KUKA KRL program: rebar_install.src

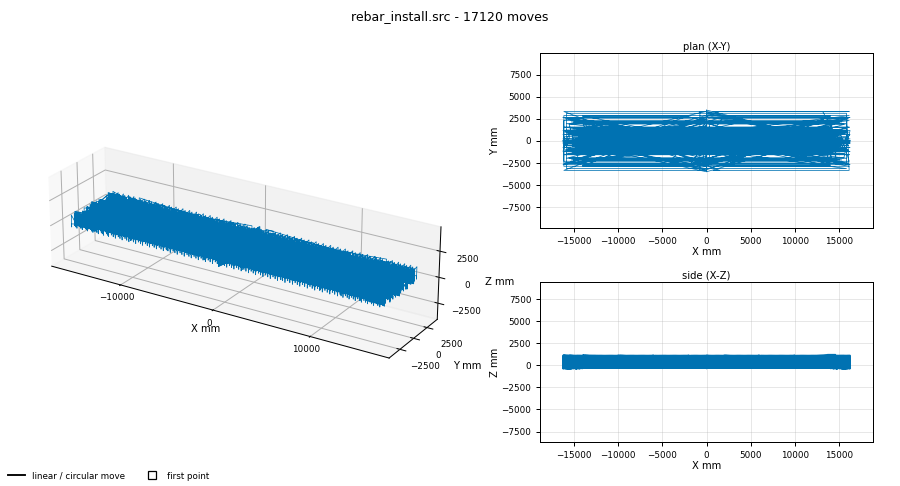
[picture p0: tool path of rebar_install.src, 17120 of 17120 moves have a stored position in this frame; points joined in program order, loops and branches not executed]
&ACCESS RVP
&REL 1
DEF REBAR_INSTALL()
  BAS(#INITMOV,0)
  ; Step 1, bar 1959
  LIN {X 14090.487,Y -1470.303,Z 792.693,A -175.02391,B 0.00000,C -180.00000} ; outside
  LIN {X 14090.487,Y -1470.303,Z -163.061,A -175.02391,B 0.00000,C -180.00000} ; preinsert
  LIN {X 14090.487,Y -1470.303,Z -413.061,A -175.02391,B 0.00000,C -180.00000} ; insert
  LIN {X 14090.487,Y -1470.303,Z -413.061,A -175.02391,B 0.00000,C -180.00000} ; release
  LIN {X 14090.487,Y -1470.303,Z -113.061,A -175.02391,B 0.00000,C -180.00000} ; retreat
  ; Step 2, bar 1960
  LIN {X 14090.487,Y 1470.303,Z 792.693,A 175.02391,B 0.00000,C 180.00000} ; outside
  LIN {X 14090.487,Y 1470.303,Z -163.061,A 175.02391,B 0.00000,C 180.00000} ; preinsert
  LIN {X 14090.487,Y 1470.303,Z -413.061,A 175.02391,B 0.00000,C 180.00000} ; insert
  LIN {X 14090.487,Y 1470.303,Z -413.061,A 175.02391,B 0.00000,C 180.00000} ; release
  LIN {X 14090.487,Y 1470.303,Z -113.061,A 175.02391,B 0.00000,C 180.00000} ; retreat
  ; Step 3, bar 1961
  LIN {X -14090.487,Y -1470.303,Z 792.693,A -4.97609,B 0.00000,C 180.00000} ; outside
  LIN {X -14090.487,Y -1470.303,Z -163.061,A -4.97609,B 0.00000,C 180.00000} ; preinsert
  LIN {X -14090.487,Y -1470.303,Z -413.061,A -4.97609,B 0.00000,C 180.00000} ; insert
  LIN {X -14090.487,Y -1470.303,Z -413.061,A -4.97609,B 0.00000,C 180.00000} ; release
  LIN {X -14090.487,Y -1470.303,Z -113.061,A -4.97609,B 0.00000,C 180.00000} ; retreat
  ; Step 4, bar 1962
  LIN {X -14090.487,Y 1470.303,Z 792.693,A 4.97609,B 0.00000,C 180.00000} ; outside
  LIN {X -14090.487,Y 1470.303,Z -163.061,A 4.97609,B 0.00000,C 180.00000} ; preinsert
  LIN {X -14090.487,Y 1470.303,Z -413.061,A 4.97609,B 0.00000,C 180.00000} ; insert
  LIN {X -14090.487,Y 1470.303,Z -413.061,A 4.97609,B 0.00000,C 180.00000} ; release
  LIN {X -14090.487,Y 1470.303,Z -113.061,A 4.97609,B 0.00000,C 180.00000} ; retreat
  ; Step 5, bar 1954
  LIN {X 0.000,Y -1540.000,Z 792.630,A 0.00000,B 0.00000,C 180.00000} ; outside
  LIN {X 0.000,Y -1540.000,Z -156.000,A 0.00000,B 0.00000,C 180.00000} ; preinsert
  LIN {X 0.000,Y -1540.000,Z -406.000,A 0.00000,B 0.00000,C 180.00000} ; insert
  LIN {X 0.000,Y -1540.000,Z -406.000,A 0.00000,B 0.00000,C 180.00000} ; release
  LIN {X 0.000,Y -1540.000,Z -106.000,A 0.00000,B 0.00000,C 180.00000} ; retreat
  ; Step 6, bar 1949
  LIN {X 0.000,Y 1540.000,Z 792.630,A 0.00000,B 0.00000,C 180.00000} ; outside
  LIN {X 0.000,Y 1540.000,Z -156.000,A 0.00000,B 0.00000,C 180.00000} ; preinsert
  LIN {X 0.000,Y 1540.000,Z -406.000,A 0.00000,B 0.00000,C 180.00000} ; insert
  LIN {X 0.000,Y 1540.000,Z -406.000,A 0.00000,B 0.00000,C 180.00000} ; release
  LIN {X 0.000,Y 1540.000,Z -106.000,A 0.00000,B 0.00000,C 180.00000} ; retreat
  ; Step 7, bar 1859
  LIN {X 0.000,Y -1752.282,Z 792.630,A 0.00000,B 0.00000,C 180.00000} ; outside
  LIN {X 0.000,Y -1752.282,Z -151.145,A 0.00000,B 0.00000,C 180.00000} ; preinsert
  LIN {X 0.000,Y -1752.282,Z -401.145,A 0.00000,B 0.00000,C 180.00000} ; insert
  LIN {X 0.000,Y -1752.282,Z -401.145,A 0.00000,B 0.00000,C 180.00000} ; release
  LIN {X 0.000,Y -1752.282,Z -101.145,A 0.00000,B 0.00000,C 180.00000} ; retreat
  ; Step 8, bar 1926
  LIN {X 0.000,Y -1632.282,Z 792.630,A 0.00000,B 0.00000,C 180.00000} ; outside
  LIN {X 0.000,Y -1632.282,Z -151.145,A 0.00000,B 0.00000,C 180.00000} ; preinsert
  LIN {X 0.000,Y -1632.282,Z -401.145,A 0.00000,B 0.00000,C 180.00000} ; insert
  LIN {X 0.000,Y -1632.282,Z -401.145,A 0.00000,B 0.00000,C 180.00000} ; release
  LIN {X 0.000,Y -1632.282,Z -101.145,A 0.00000,B 0.00000,C 180.00000} ; retreat
  ; Step 9, bar 1925
  LIN {X 0.000,Y 1632.282,Z 792.630,A 0.00000,B 0.00000,C 180.00000} ; outside
  LIN {X 0.000,Y 1632.282,Z -151.145,A 0.00000,B 0.00000,C 180.00000} ; preinsert
  LIN {X 0.000,Y 1632.282,Z -401.145,A 0.00000,B 0.00000,C 180.00000} ; insert
  LIN {X 0.000,Y 1632.282,Z -401.145,A 0.00000,B 0.00000,C 180.00000} ; release
  LIN {X 0.000,Y 1632.282,Z -101.145,A 0.00000,B 0.00000,C 180.00000} ; retreat
  ; Step 10, bar 1872
  LIN {X 0.000,Y 1752.282,Z 792.630,A 0.00000,B 0.00000,C 180.00000} ; outside
  LIN {X 0.000,Y 1752.282,Z -151.145,A 0.00000,B 0.00000,C 180.00000} ; preinsert
  LIN {X 0.000,Y 1752.282,Z -401.145,A 0.00000,B 0.00000,C 180.00000} ; insert
  LIN {X 0.000,Y 1752.282,Z -401.145,A 0.00000,B 0.00000,C 180.00000} ; release
  LIN {X 0.000,Y 1752.282,Z -101.145,A 0.00000,B 0.00000,C 180.00000} ; retreat
  ; Step 11, bar 3422
  LIN {X -16169.500,Y -1557.401,Z 792.630,A 90.00000,B 0.00000,C 180.00000} ; outside
  LIN {X -16169.500,Y -1557.401,Z -142.000,A 90.00000,B 0.00000,C 180.00000} ; preinsert
  LIN {X -16169.500,Y -1557.401,Z -392.000,A 90.00000,B 0.00000,C 180.00000} ; insert
  LIN {X -16169.500,Y -1557.401,Z -392.000,A 90.00000,B 0.00000,C 180.00000} ; release
  LIN {X -16169.500,Y -1557.401,Z -92.000,A 90.00000,B 0.00000,C 180.00000} ; retreat
  ; Step 12, bar 3418
  LIN {X 16169.500,Y -1557.401,Z 792.630,A 90.00000,B 0.00000,C 180.00000} ; outside
  LIN {X 16169.500,Y -1557.401,Z -142.000,A 90.00000,B 0.00000,C 180.00000} ; preinsert
  LIN {X 16169.500,Y -1557.401,Z -392.000,A 90.00000,B 0.00000,C 180.00000} ; insert
  LIN {X 16169.500,Y -1557.401,Z -392.000,A 90.00000,B 0.00000,C 180.00000} ; release
  LIN {X 16169.500,Y -1557.401,Z -92.000,A 90.00000,B 0.00000,C 180.00000} ; retreat
  ; Step 13, bar 3420
  LIN {X -16169.500,Y 1557.401,Z 792.630,A -90.00000,B 0.00000,C 180.00000} ; outside
  LIN {X -16169.500,Y 1557.401,Z -142.000,A -90.00000,B 0.00000,C 180.00000} ; preinsert
  LIN {X -16169.500,Y 1557.401,Z -392.000,A -90.00000,B 0.00000,C 180.00000} ; insert
  LIN {X -16169.500,Y 1557.401,Z -392.000,A -90.00000,B 0.00000,C 180.00000} ; release
  LIN {X -16169.500,Y 1557.401,Z -92.000,A -90.00000,B 0.00000,C 180.00000} ; retreat
  ; Step 14, bar 3416
  LIN {X 16169.500,Y 1557.401,Z 792.630,A -90.00000,B 0.00000,C 180.00000} ; outside
  LIN {X 16169.500,Y 1557.401,Z -142.000,A -90.00000,B 0.00000,C 180.00000} ; preinsert
  LIN {X 16169.500,Y 1557.401,Z -392.000,A -90.00000,B 0.00000,C 180.00000} ; insert
  LIN {X 16169.500,Y 1557.401,Z -392.000,A -90.00000,B 0.00000,C 180.00000} ; release
  LIN {X 16169.500,Y 1557.401,Z -92.000,A -90.00000,B 0.00000,C 180.00000} ; retreat
  ; Step 15, bar 1860
  LIN {X 0.000,Y -1977.000,Z 792.630,A 0.00000,B 0.00000,C 180.00000} ; outside
  LIN {X 0.000,Y -1977.000,Z -124.093,A 0.00000,B 0.00000,C 180.00000} ; preinsert
  LIN {X 0.000,Y -1977.000,Z -374.093,A 0.00000,B 0.00000,C 180.00000} ; insert
  LIN {X 0.000,Y -1977.000,Z -374.093,A 0.00000,B 0.00000,C 180.00000} ; release
  LIN {X 0.000,Y -1977.000,Z -74.093,A 0.00000,B 0.00000,C 180.00000} ; retreat
  ; Step 16, bar 1873
  LIN {X 0.000,Y 1977.000,Z 792.630,A 0.00000,B 0.00000,C 180.00000} ; outside
  LIN {X 0.000,Y 1977.000,Z -124.093,A 0.00000,B 0.00000,C 180.00000} ; preinsert
  LIN {X 0.000,Y 1977.000,Z -374.093,A 0.00000,B 0.00000,C 180.00000} ; insert
  LIN {X 0.000,Y 1977.000,Z -374.093,A 0.00000,B 0.00000,C 180.00000} ; release
  LIN {X 0.000,Y 1977.000,Z -74.093,A 0.00000,B 0.00000,C 180.00000} ; retreat
  ; Step 17, bar 1953
  LIN {X 0.000,Y -1420.000,Z 792.630,A 0.00000,B 0.00000,C 180.00000} ; outside
  LIN {X 0.000,Y -1420.000,Z -118.500,A 0.00000,B 0.00000,C 180.00000} ; preinsert
  LIN {X 0.000,Y -1420.000,Z -368.500,A 0.00000,B 0.00000,C 180.00000} ; insert
  LIN {X 0.000,Y -1420.000,Z -368.500,A 0.00000,B 0.00000,C 180.00000} ; release
  LIN {X 0.000,Y -1420.000,Z -68.500,A 0.00000,B 0.00000,C 180.00000} ; retreat
  ; Step 18, bar 1948
  LIN {X 0.000,Y 1420.000,Z 792.630,A 0.00000,B 0.00000,C 180.00000} ; outside
  LIN {X 0.000,Y 1420.000,Z -118.500,A 0.00000,B 0.00000,C 180.00000} ; preinsert
  LIN {X 0.000,Y 1420.000,Z -368.500,A 0.00000,B 0.00000,C 180.00000} ; insert
  LIN {X 0.000,Y 1420.000,Z -368.500,A 0.00000,B 0.00000,C 180.00000} ; release
  LIN {X 0.000,Y 1420.000,Z -68.500,A 0.00000,B 0.00000,C 180.00000} ; retreat
  ; Step 19, bar 3289
  LIN {X -15485.187,Y -1114.878,Z 792.759,A -134.96824,B 0.00000,C -180.00000} ; outside
  LIN {X -15485.187,Y -1114.878,Z -98.768,A -134.96824,B 0.00000,C -180.00000} ; preinsert
  LIN {X -15485.187,Y -1114.878,Z -348.768,A -134.96824,B 0.00000,C -180.00000} ; insert
  LIN {X -15485.187,Y -1114.878,Z -348.768,A -134.96824,B 0.00000,C -180.00000} ; release
  LIN {X -15485.187,Y -1114.878,Z -48.768,A -134.96824,B 0.00000,C -180.00000} ; retreat
  ; Step 20, bar 3291
  LIN {X -15614.813,Y -1114.878,Z 792.759,A -45.03176,B 0.00000,C 180.00000} ; outside
  LIN {X -15614.813,Y -1114.878,Z -98.768,A -45.03176,B 0.00000,C 180.00000} ; preinsert
  LIN {X -15614.813,Y -1114.878,Z -348.768,A -45.03176,B 0.00000,C 180.00000} ; insert
  LIN {X -15614.813,Y -1114.878,Z -348.768,A -45.03176,B 0.00000,C 180.00000} ; release
  LIN {X -15614.813,Y -1114.878,Z -48.768,A -45.03176,B 0.00000,C 180.00000} ; retreat
  ; Step 21, bar 3369
  LIN {X 15485.187,Y -1114.878,Z 792.759,A -45.03176,B 0.00000,C 180.00000} ; outside
  LIN {X 15485.187,Y -1114.878,Z -98.768,A -45.03176,B 0.00000,C 180.00000} ; preinsert
  LIN {X 15485.187,Y -1114.878,Z -348.768,A -45.03176,B 0.00000,C 180.00000} ; insert
  LIN {X 15485.187,Y -1114.878,Z -348.768,A -45.03176,B 0.00000,C 180.00000} ; release
  LIN {X 15485.187,Y -1114.878,Z -48.768,A -45.03176,B 0.00000,C 180.00000} ; retreat
  ; Step 22, bar 3371
  LIN {X 15614.813,Y -1114.878,Z 792.759,A -134.96824,B 0.00000,C -180.00000} ; outside
  LIN {X 15614.813,Y -1114.878,Z -98.768,A -134.96824,B 0.00000,C -180.00000} ; preinsert
  LIN {X 15614.813,Y -1114.878,Z -348.768,A -134.96824,B 0.00000,C -180.00000} ; insert
  LIN {X 15614.813,Y -1114.878,Z -348.768,A -134.96824,B 0.00000,C -180.00000} ; release
  LIN {X 15614.813,Y -1114.878,Z -48.768,A -134.96824,B 0.00000,C -180.00000} ; retreat
  ; Step 23, bar 3290
  LIN {X -15485.122,Y -985.187,Z 792.759,A -44.96824,B 0.00000,C 180.00000} ; outside
  LIN {X -15485.122,Y -985.187,Z -98.768,A -44.96824,B 0.00000,C 180.00000} ; preinsert
  LIN {X -15485.122,Y -985.187,Z -348.768,A -44.96824,B 0.00000,C 180.00000} ; insert
  LIN {X -15485.122,Y -985.187,Z -348.768,A -44.96824,B 0.00000,C 180.00000} ; release
  LIN {X -15485.122,Y -985.187,Z -48.768,A -44.96824,B 0.00000,C 180.00000} ; retreat
  ; Step 24, bar 3288
  LIN {X -15614.878,Y -985.187,Z 792.759,A -135.03176,B 0.00000,C -180.00000} ; outside
  LIN {X -15614.878,Y -985.187,Z -98.768,A -135.03176,B 0.00000,C -180.00000} ; preinsert
  LIN {X -15614.878,Y -985.187,Z -348.768,A -135.03176,B 0.00000,C -180.00000} ; insert
  LIN {X -15614.878,Y -985.187,Z -348.768,A -135.03176,B 0.00000,C -180.00000} ; release
  LIN {X -15614.878,Y -985.187,Z -48.768,A -135.03176,B 0.00000,C -180.00000} ; retreat
  ; Step 25, bar 3370
  LIN {X 15485.122,Y -985.187,Z 792.759,A -135.03176,B 0.00000,C 180.00000} ; outside
  LIN {X 15485.122,Y -985.187,Z -98.768,A -135.03176,B 0.00000,C 180.00000} ; preinsert
  LIN {X 15485.122,Y -985.187,Z -348.768,A -135.03176,B 0.00000,C 180.00000} ; insert
  LIN {X 15485.122,Y -985.187,Z -348.768,A -135.03176,B 0.00000,C 180.00000} ; release
  LIN {X 15485.122,Y -985.187,Z -48.768,A -135.03176,B 0.00000,C 180.00000} ; retreat
  ; Step 26, bar 3368
  LIN {X 15614.878,Y -985.187,Z 792.759,A -44.96824,B 0.00000,C 180.00000} ; outside
  LIN {X 15614.878,Y -985.187,Z -98.768,A -44.96824,B 0.00000,C 180.00000} ; preinsert
  LIN {X 15614.878,Y -985.187,Z -348.768,A -44.96824,B 0.00000,C 180.00000} ; insert
  LIN {X 15614.878,Y -985.187,Z -348.768,A -44.96824,B 0.00000,C 180.00000} ; release
  LIN {X 15614.878,Y -985.187,Z -48.768,A -44.96824,B 0.00000,C 180.00000} ; retreat
  ; Step 27, bar 3328
  LIN {X -15614.878,Y 985.187,Z 792.759,A 135.03176,B 0.00000,C 180.00000} ; outside
  LIN {X -15614.878,Y 985.187,Z -98.768,A 135.03176,B 0.00000,C 180.00000} ; preinsert
  LIN {X -15614.878,Y 985.187,Z -348.768,A 135.03176,B 0.00000,C 180.00000} ; insert
  LIN {X -15614.878,Y 985.187,Z -348.768,A 135.03176,B 0.00000,C 180.00000} ; release
  LIN {X -15614.878,Y 985.187,Z -48.768,A 135.03176,B 0.00000,C 180.00000} ; retreat
  ; Step 28, bar 3408
  LIN {X 15614.878,Y 985.187,Z 792.759,A 44.96824,B 0.00000,C 180.00000} ; outside
  LIN {X 15614.878,Y 985.187,Z -98.768,A 44.96824,B 0.00000,C 180.00000} ; preinsert
  LIN {X 15614.878,Y 985.187,Z -348.768,A 44.96824,B 0.00000,C 180.00000} ; insert
  LIN {X 15614.878,Y 985.187,Z -348.768,A 44.96824,B 0.00000,C 180.00000} ; release
  LIN {X 15614.878,Y 985.187,Z -48.768,A 44.96824,B 0.00000,C 180.00000} ; retreat
  ; Step 29, bar 3330
  LIN {X -15485.122,Y 985.187,Z 792.759,A 44.96824,B 0.00000,C 180.00000} ; outside
  LIN {X -15485.122,Y 985.187,Z -98.768,A 44.96824,B 0.00000,C 180.00000} ; preinsert
  LIN {X -15485.122,Y 985.187,Z -348.768,A 44.96824,B 0.00000,C 180.00000} ; insert
  LIN {X -15485.122,Y 985.187,Z -348.768,A 44.96824,B 0.00000,C 180.00000} ; release
  LIN {X -15485.122,Y 985.187,Z -48.768,A 44.96824,B 0.00000,C 180.00000} ; retreat
  ; Step 30, bar 3410
  LIN {X 15485.122,Y 985.187,Z 792.759,A 135.03176,B 0.00000,C 180.00000} ; outside
  LIN {X 15485.122,Y 985.187,Z -98.768,A 135.03176,B 0.00000,C 180.00000} ; preinsert
  LIN {X 15485.122,Y 985.187,Z -348.768,A 135.03176,B 0.00000,C 180.00000} ; insert
  LIN {X 15485.122,Y 985.187,Z -348.768,A 135.03176,B 0.00000,C 180.00000} ; release
  LIN {X 15485.122,Y 985.187,Z -48.768,A 135.03176,B 0.00000,C 180.00000} ; retreat
  ; Step 31, bar 3331
  LIN {X -15614.813,Y 1114.878,Z 792.759,A 45.03176,B 0.00000,C 180.00000} ; outside
  LIN {X -15614.813,Y 1114.878,Z -98.768,A 45.03176,B 0.00000,C 180.00000} ; preinsert
  LIN {X -15614.813,Y 1114.878,Z -348.768,A 45.03176,B 0.00000,C 180.00000} ; insert
  LIN {X -15614.813,Y 1114.878,Z -348.768,A 45.03176,B 0.00000,C 180.00000} ; release
  LIN {X -15614.813,Y 1114.878,Z -48.768,A 45.03176,B 0.00000,C 180.00000} ; retreat
  ; Step 32, bar 3411
  LIN {X 15614.813,Y 1114.878,Z 792.759,A 134.96824,B 0.00000,C 180.00000} ; outside
  LIN {X 15614.813,Y 1114.878,Z -98.768,A 134.96824,B 0.00000,C 180.00000} ; preinsert
  LIN {X 15614.813,Y 1114.878,Z -348.768,A 134.96824,B 0.00000,C 180.00000} ; insert
  LIN {X 15614.813,Y 1114.878,Z -348.768,A 134.96824,B 0.00000,C 180.00000} ; release
  LIN {X 15614.813,Y 1114.878,Z -48.768,A 134.96824,B 0.00000,C 180.00000} ; retreat
  ; Step 33, bar 3329
  LIN {X -15485.187,Y 1114.878,Z 792.759,A 134.96824,B 0.00000,C 180.00000} ; outside
  LIN {X -15485.187,Y 1114.878,Z -98.768,A 134.96824,B 0.00000,C 180.00000} ; preinsert
  LIN {X -15485.187,Y 1114.878,Z -348.768,A 134.96824,B 0.00000,C 180.00000} ; insert
  LIN {X -15485.187,Y 1114.878,Z -348.768,A 134.96824,B 0.00000,C 180.00000} ; release
  LIN {X -15485.187,Y 1114.878,Z -48.768,A 134.96824,B 0.00000,C 180.00000} ; retreat
  ; Step 34, bar 3409
  LIN {X 15485.187,Y 1114.878,Z 792.759,A 45.03176,B 0.00000,C 180.00000} ; outside
  LIN {X 15485.187,Y 1114.878,Z -98.768,A 45.03176,B 0.00000,C 180.00000} ; preinsert
  LIN {X 15485.187,Y 1114.878,Z -348.768,A 45.03176,B 0.00000,C 180.00000} ; insert
  LIN {X 15485.187,Y 1114.878,Z -348.768,A 45.03176,B 0.00000,C 180.00000} ; release
  LIN {X 15485.187,Y 1114.878,Z -48.768,A 45.03176,B 0.00000,C 180.00000} ; retreat
  ; Step 35, bar 3269
  LIN {X -14485.187,Y -1114.878,Z 792.759,A -134.96824,B 0.00000,C -180.00000} ; outside
  LIN {X -14485.187,Y -1114.878,Z -98.768,A -134.96824,B 0.00000,C -180.00000} ; preinsert
  LIN {X -14485.187,Y -1114.878,Z -348.768,A -134.96824,B 0.00000,C -180.00000} ; insert
  LIN {X -14485.187,Y -1114.878,Z -348.768,A -134.96824,B 0.00000,C -180.00000} ; release
  LIN {X -14485.187,Y -1114.878,Z -48.768,A -134.96824,B 0.00000,C -180.00000} ; retreat
  ; Step 36, bar 3271
  LIN {X -14614.813,Y -1114.878,Z 792.759,A -45.03176,B 0.00000,C 180.00000} ; outside
  LIN {X -14614.813,Y -1114.878,Z -98.768,A -45.03176,B 0.00000,C 180.00000} ; preinsert
  LIN {X -14614.813,Y -1114.878,Z -348.768,A -45.03176,B 0.00000,C 180.00000} ; insert
  LIN {X -14614.813,Y -1114.878,Z -348.768,A -45.03176,B 0.00000,C 180.00000} ; release
  LIN {X -14614.813,Y -1114.878,Z -48.768,A -45.03176,B 0.00000,C 180.00000} ; retreat
  ; Step 37, bar 3349
  LIN {X 14485.187,Y -1114.878,Z 792.759,A -45.03176,B 0.00000,C 180.00000} ; outside
  LIN {X 14485.187,Y -1114.878,Z -98.768,A -45.03176,B 0.00000,C 180.00000} ; preinsert
  LIN {X 14485.187,Y -1114.878,Z -348.768,A -45.03176,B 0.00000,C 180.00000} ; insert
  LIN {X 14485.187,Y -1114.878,Z -348.768,A -45.03176,B 0.00000,C 180.00000} ; release
  LIN {X 14485.187,Y -1114.878,Z -48.768,A -45.03176,B 0.00000,C 180.00000} ; retreat
  ; Step 38, bar 3351
  LIN {X 14614.813,Y -1114.878,Z 792.759,A -134.96824,B 0.00000,C -180.00000} ; outside
  LIN {X 14614.813,Y -1114.878,Z -98.768,A -134.96824,B 0.00000,C -180.00000} ; preinsert
  LIN {X 14614.813,Y -1114.878,Z -348.768,A -134.96824,B 0.00000,C -180.00000} ; insert
  LIN {X 14614.813,Y -1114.878,Z -348.768,A -134.96824,B 0.00000,C -180.00000} ; release
  LIN {X 14614.813,Y -1114.878,Z -48.768,A -134.96824,B 0.00000,C -180.00000} ; retreat
  ; Step 39, bar 3270
  LIN {X -14485.122,Y -985.187,Z 792.759,A -44.96824,B 0.00000,C 180.00000} ; outside
  LIN {X -14485.122,Y -985.187,Z -98.768,A -44.96824,B 0.00000,C 180.00000} ; preinsert
  LIN {X -14485.122,Y -985.187,Z -348.768,A -44.96824,B 0.00000,C 180.00000} ; insert
  LIN {X -14485.122,Y -985.187,Z -348.768,A -44.96824,B 0.00000,C 180.00000} ; release
  LIN {X -14485.122,Y -985.187,Z -48.768,A -44.96824,B 0.00000,C 180.00000} ; retreat
  ; Step 40, bar 3268
  LIN {X -14614.878,Y -985.187,Z 792.759,A -135.03176,B 0.00000,C -180.00000} ; outside
  LIN {X -14614.878,Y -985.187,Z -98.768,A -135.03176,B 0.00000,C -180.00000} ; preinsert
  LIN {X -14614.878,Y -985.187,Z -348.768,A -135.03176,B 0.00000,C -180.00000} ; insert
  LIN {X -14614.878,Y -985.187,Z -348.768,A -135.03176,B 0.00000,C -180.00000} ; release
  LIN {X -14614.878,Y -985.187,Z -48.768,A -135.03176,B 0.00000,C -180.00000} ; retreat
  ; Step 41, bar 3350
  LIN {X 14485.122,Y -985.187,Z 792.759,A -135.03176,B 0.00000,C 180.00000} ; outside
  LIN {X 14485.122,Y -985.187,Z -98.768,A -135.03176,B 0.00000,C 180.00000} ; preinsert
  LIN {X 14485.122,Y -985.187,Z -348.768,A -135.03176,B 0.00000,C 180.00000} ; insert
  LIN {X 14485.122,Y -985.187,Z -348.768,A -135.03176,B 0.00000,C 180.00000} ; release
  LIN {X 14485.122,Y -985.187,Z -48.768,A -135.03176,B 0.00000,C 180.00000} ; retreat
  ; Step 42, bar 3348
  LIN {X 14614.878,Y -985.187,Z 792.759,A -44.96824,B 0.00000,C 180.00000} ; outside
  LIN {X 14614.878,Y -985.187,Z -98.768,A -44.96824,B 0.00000,C 180.00000} ; preinsert
  LIN {X 14614.878,Y -985.187,Z -348.768,A -44.96824,B 0.00000,C 180.00000} ; insert
  LIN {X 14614.878,Y -985.187,Z -348.768,A -44.96824,B 0.00000,C 180.00000} ; release
  LIN {X 14614.878,Y -985.187,Z -48.768,A -44.96824,B 0.00000,C 180.00000} ; retreat
  ; Step 43, bar 3308
  LIN {X -14614.878,Y 985.187,Z 792.759,A 135.03176,B 0.00000,C 180.00000} ; outside
  LIN {X -14614.878,Y 985.187,Z -98.768,A 135.03176,B 0.00000,C 180.00000} ; preinsert
  LIN {X -14614.878,Y 985.187,Z -348.768,A 135.03176,B 0.00000,C 180.00000} ; insert
  LIN {X -14614.878,Y 985.187,Z -348.768,A 135.03176,B 0.00000,C 180.00000} ; release
  LIN {X -14614.878,Y 985.187,Z -48.768,A 135.03176,B 0.00000,C 180.00000} ; retreat
  ; Step 44, bar 3388
  LIN {X 14614.878,Y 985.187,Z 792.759,A 44.96824,B 0.00000,C 180.00000} ; outside
  LIN {X 14614.878,Y 985.187,Z -98.768,A 44.96824,B 0.00000,C 180.00000} ; preinsert
  LIN {X 14614.878,Y 985.187,Z -348.768,A 44.96824,B 0.00000,C 180.00000} ; insert
  LIN {X 14614.878,Y 985.187,Z -348.768,A 44.96824,B 0.00000,C 180.00000} ; release
  LIN {X 14614.878,Y 985.187,Z -48.768,A 44.96824,B 0.00000,C 180.00000} ; retreat
  ; Step 45, bar 3310
  LIN {X -14485.122,Y 985.187,Z 792.759,A 44.96824,B 0.00000,C 180.00000} ; outside
  LIN {X -14485.122,Y 985.187,Z -98.768,A 44.96824,B 0.00000,C 180.00000} ; preinsert
  LIN {X -14485.122,Y 985.187,Z -348.768,A 44.96824,B 0.00000,C 180.00000} ; insert
  LIN {X -14485.122,Y 985.187,Z -348.768,A 44.96824,B 0.00000,C 180.00000} ; release
  LIN {X -14485.122,Y 985.187,Z -48.768,A 44.96824,B 0.00000,C 180.00000} ; retreat
  ; Step 46, bar 3390
  LIN {X 14485.122,Y 985.187,Z 792.759,A 135.03176,B 0.00000,C 180.00000} ; outside
  LIN {X 14485.122,Y 985.187,Z -98.768,A 135.03176,B 0.00000,C 180.00000} ; preinsert
  LIN {X 14485.122,Y 985.187,Z -348.768,A 135.03176,B 0.00000,C 180.00000} ; insert
  LIN {X 14485.122,Y 985.187,Z -348.768,A 135.03176,B 0.00000,C 180.00000} ; release
  LIN {X 14485.122,Y 985.187,Z -48.768,A 135.03176,B 0.00000,C 180.00000} ; retreat
  ; Step 47, bar 3311
  LIN {X -14614.813,Y 1114.878,Z 792.759,A 45.03176,B 0.00000,C 180.00000} ; outside
  LIN {X -14614.813,Y 1114.878,Z -98.768,A 45.03176,B 0.00000,C 180.00000} ; preinsert
  LIN {X -14614.813,Y 1114.878,Z -348.768,A 45.03176,B 0.00000,C 180.00000} ; insert
  LIN {X -14614.813,Y 1114.878,Z -348.768,A 45.03176,B 0.00000,C 180.00000} ; release
  LIN {X -14614.813,Y 1114.878,Z -48.768,A 45.03176,B 0.00000,C 180.00000} ; retreat
  ; Step 48, bar 3391
  LIN {X 14614.813,Y 1114.878,Z 792.759,A 134.96824,B 0.00000,C 180.00000} ; outside
  LIN {X 14614.813,Y 1114.878,Z -98.768,A 134.96824,B 0.00000,C 180.00000} ; preinsert
  LIN {X 14614.813,Y 1114.878,Z -348.768,A 134.96824,B 0.00000,C 180.00000} ; insert
  LIN {X 14614.813,Y 1114.878,Z -348.768,A 134.96824,B 0.00000,C 180.00000} ; release
  LIN {X 14614.813,Y 1114.878,Z -48.768,A 134.96824,B 0.00000,C 180.00000} ; retreat
  ; Step 49, bar 3309
  LIN {X -14485.187,Y 1114.878,Z 792.759,A 134.96824,B 0.00000,C 180.00000} ; outside
  LIN {X -14485.187,Y 1114.878,Z -98.768,A 134.96824,B 0.00000,C 180.00000} ; preinsert
  LIN {X -14485.187,Y 1114.878,Z -348.768,A 134.96824,B 0.00000,C 180.00000} ; insert
  LIN {X -14485.187,Y 1114.878,Z -348.768,A 134.96824,B 0.00000,C 180.00000} ; release
  LIN {X -14485.187,Y 1114.878,Z -48.768,A 134.96824,B 0.00000,C 180.00000} ; retreat
  ; Step 50, bar 3389
  LIN {X 14485.187,Y 1114.878,Z 792.759,A 45.03176,B 0.00000,C 180.00000} ; outside
  LIN {X 14485.187,Y 1114.878,Z -98.768,A 45.03176,B 0.00000,C 180.00000} ; preinsert
  LIN {X 14485.187,Y 1114.878,Z -348.768,A 45.03176,B 0.00000,C 180.00000} ; insert
  LIN {X 14485.187,Y 1114.878,Z -348.768,A 45.03176,B 0.00000,C 180.00000} ; release
  LIN {X 14485.187,Y 1114.878,Z -48.768,A 45.03176,B 0.00000,C 180.00000} ; retreat
  ; Step 51, bar 1952
  LIN {X 0.000,Y -1325.000,Z 792.630,A 0.00000,B 0.00000,C 180.00000} ; outside
  LIN {X 0.000,Y -1325.000,Z -89.125,A 0.00000,B 0.00000,C 180.00000} ; preinsert
  LIN {X 0.000,Y -1325.000,Z -339.125,A 0.00000,B 0.00000,C 180.00000} ; insert
  LIN {X 0.000,Y -1325.000,Z -339.125,A 0.00000,B 0.00000,C 180.00000} ; release
  LIN {X 0.000,Y -1325.000,Z -39.125,A 0.00000,B 0.00000,C 180.00000} ; retreat
  ; Step 52, bar 1947
  LIN {X 0.000,Y 1325.000,Z 792.630,A 0.00000,B 0.00000,C 180.00000} ; outside
  LIN {X 0.000,Y 1325.000,Z -89.125,A 0.00000,B 0.00000,C 180.00000} ; preinsert
  LIN {X 0.000,Y 1325.000,Z -339.125,A 0.00000,B 0.00000,C 180.00000} ; insert
  LIN {X 0.000,Y 1325.000,Z -339.125,A 0.00000,B 0.00000,C 180.00000} ; release
  LIN {X 0.000,Y 1325.000,Z -39.125,A 0.00000,B 0.00000,C 180.00000} ; retreat
  ; Step 53, bar 3282
  LIN {X -15779.028,Y -1023.446,Z 793.100,A -89.93308,B 0.00000,C 180.00000} ; outside
  LIN {X -15779.028,Y -1023.446,Z -156.648,A -89.93308,B 0.00000,C 180.00000} ; preinsert
  LIN {X -15779.028,Y -1023.446,Z -406.648,A -89.93308,B 0.00000,C 180.00000} ; insert
  LIN {X -15779.028,Y -1023.446,Z -406.648,A -89.93308,B 0.00000,C 180.00000} ; release
  LIN {X -15779.028,Y -1023.446,Z -106.648,A -89.93308,B 0.00000,C 180.00000} ; retreat
  ; Step 54, bar 3278
  LIN {X -15395.940,Y -1023.446,Z 793.100,A -89.99904,B 0.00000,C 180.00000} ; outside
  LIN {X -15395.940,Y -1023.446,Z -156.648,A -89.99904,B 0.00000,C 180.00000} ; preinsert
  LIN {X -15395.940,Y -1023.446,Z -406.648,A -89.99904,B 0.00000,C 180.00000} ; insert
  LIN {X -15395.940,Y -1023.446,Z -406.648,A -89.99904,B 0.00000,C 180.00000} ; release
  LIN {X -15395.940,Y -1023.446,Z -106.648,A -89.99904,B 0.00000,C 180.00000} ; retreat
  ; Step 55, bar 3279
  LIN {X -15320.940,Y -1023.446,Z 793.100,A -89.99904,B 0.00000,C 180.00000} ; outside
  LIN {X -15320.940,Y -1023.446,Z -156.648,A -89.99904,B 0.00000,C 180.00000} ; preinsert
  LIN {X -15320.940,Y -1023.446,Z -406.648,A -89.99904,B 0.00000,C 180.00000} ; insert
  LIN {X -15320.940,Y -1023.446,Z -406.648,A -89.99904,B 0.00000,C 180.00000} ; release
  LIN {X -15320.940,Y -1023.446,Z -106.648,A -89.99904,B 0.00000,C 180.00000} ; retreat
  ; Step 56, bar 3359
  LIN {X 15320.972,Y -1023.446,Z 793.100,A -89.93308,B 0.00000,C 180.00000} ; outside
  LIN {X 15320.972,Y -1023.446,Z -156.648,A -89.93308,B 0.00000,C 180.00000} ; preinsert
  LIN {X 15320.972,Y -1023.446,Z -406.648,A -89.93308,B 0.00000,C 180.00000} ; insert
  LIN {X 15320.972,Y -1023.446,Z -406.648,A -89.93308,B 0.00000,C 180.00000} ; release
  LIN {X 15320.972,Y -1023.446,Z -106.648,A -89.93308,B 0.00000,C 180.00000} ; retreat
  ; Step 57, bar 3358
  LIN {X 15395.972,Y -1023.446,Z 793.100,A -89.93308,B 0.00000,C 180.00000} ; outside
  LIN {X 15395.972,Y -1023.446,Z -156.648,A -89.93308,B 0.00000,C 180.00000} ; preinsert
  LIN {X 15395.972,Y -1023.446,Z -406.648,A -89.93308,B 0.00000,C 180.00000} ; insert
  LIN {X 15395.972,Y -1023.446,Z -406.648,A -89.93308,B 0.00000,C 180.00000} ; release
  LIN {X 15395.972,Y -1023.446,Z -106.648,A -89.93308,B 0.00000,C 180.00000} ; retreat
  ; Step 58, bar 3362
  LIN {X 15779.060,Y -1023.446,Z 793.100,A -89.99904,B 0.00000,C 180.00000} ; outside
  LIN {X 15779.060,Y -1023.446,Z -156.648,A -89.99904,B 0.00000,C 180.00000} ; preinsert
  LIN {X 15779.060,Y -1023.446,Z -406.648,A -89.99904,B 0.00000,C 180.00000} ; insert
  LIN {X 15779.060,Y -1023.446,Z -406.648,A -89.99904,B 0.00000,C 180.00000} ; release
  LIN {X 15779.060,Y -1023.446,Z -106.648,A -89.99904,B 0.00000,C 180.00000} ; retreat
  ; Step 59, bar 3322
  LIN {X -15779.060,Y 1023.446,Z 793.100,A 90.00096,B 0.00000,C 180.00000} ; outside
  LIN {X -15779.060,Y 1023.446,Z -156.648,A 90.00096,B 0.00000,C 180.00000} ; preinsert
  LIN {X -15779.060,Y 1023.446,Z -406.648,A 90.00096,B 0.00000,C 180.00000} ; insert
  LIN {X -15779.060,Y 1023.446,Z -406.648,A 90.00096,B 0.00000,C 180.00000} ; release
  LIN {X -15779.060,Y 1023.446,Z -106.648,A 90.00096,B 0.00000,C 180.00000} ; retreat
  ; Step 60, bar 3318
  LIN {X -15395.972,Y 1023.446,Z 793.100,A 90.06692,B 0.00000,C 180.00000} ; outside
  LIN {X -15395.972,Y 1023.446,Z -156.648,A 90.06692,B 0.00000,C 180.00000} ; preinsert
  LIN {X -15395.972,Y 1023.446,Z -406.648,A 90.06692,B 0.00000,C 180.00000} ; insert
  LIN {X -15395.972,Y 1023.446,Z -406.648,A 90.06692,B 0.00000,C 180.00000} ; release
  LIN {X -15395.972,Y 1023.446,Z -106.648,A 90.06692,B 0.00000,C 180.00000} ; retreat
  ; Step 61, bar 3319
  LIN {X -15320.972,Y 1023.446,Z 793.100,A 90.06692,B 0.00000,C 180.00000} ; outside
  LIN {X -15320.972,Y 1023.446,Z -156.648,A 90.06692,B 0.00000,C 180.00000} ; preinsert
  LIN {X -15320.972,Y 1023.446,Z -406.648,A 90.06692,B 0.00000,C 180.00000} ; insert
  LIN {X -15320.972,Y 1023.446,Z -406.648,A 90.06692,B 0.00000,C 180.00000} ; release
  LIN {X -15320.972,Y 1023.446,Z -106.648,A 90.06692,B 0.00000,C 180.00000} ; retreat
  ; Step 62, bar 3399
  LIN {X 15320.940,Y 1023.446,Z 793.100,A 90.00096,B 0.00000,C 180.00000} ; outside
  LIN {X 15320.940,Y 1023.446,Z -156.648,A 90.00096,B 0.00000,C 180.00000} ; preinsert
  LIN {X 15320.940,Y 1023.446,Z -406.648,A 90.00096,B 0.00000,C 180.00000} ; insert
  LIN {X 15320.940,Y 1023.446,Z -406.648,A 90.00096,B 0.00000,C 180.00000} ; release
  LIN {X 15320.940,Y 1023.446,Z -106.648,A 90.00096,B 0.00000,C 180.00000} ; retreat
  ; Step 63, bar 3398
  LIN {X 15395.940,Y 1023.446,Z 793.100,A 90.00096,B 0.00000,C 180.00000} ; outside
  LIN {X 15395.940,Y 1023.446,Z -156.648,A 90.00096,B 0.00000,C 180.00000} ; preinsert
  LIN {X 15395.940,Y 1023.446,Z -406.648,A 90.00096,B 0.00000,C 180.00000} ; insert
  LIN {X 15395.940,Y 1023.446,Z -406.648,A 90.00096,B 0.00000,C 180.00000} ; release
  LIN {X 15395.940,Y 1023.446,Z -106.648,A 90.00096,B 0.00000,C 180.00000} ; retreat
  ; Step 64, bar 3402
  LIN {X 15779.028,Y 1023.446,Z 793.100,A 90.06692,B 0.00000,C 180.00000} ; outside
  LIN {X 15779.028,Y 1023.446,Z -156.648,A 90.06692,B 0.00000,C 180.00000} ; preinsert
  LIN {X 15779.028,Y 1023.446,Z -406.648,A 90.06692,B 0.00000,C 180.00000} ; insert
  LIN {X 15779.028,Y 1023.446,Z -406.648,A 90.06692,B 0.00000,C 180.00000} ; release
  LIN {X 15779.028,Y 1023.446,Z -106.648,A 90.06692,B 0.00000,C 180.00000} ; retreat
  ; Step 65, bar 3283
  LIN {X -15854.028,Y -1023.446,Z 793.100,A -89.93308,B 0.00000,C 180.00000} ; outside
  LIN {X -15854.028,Y -1023.446,Z -156.648,A -89.93308,B 0.00000,C 180.00000} ; preinsert
  LIN {X -15854.028,Y -1023.446,Z -406.648,A -89.93308,B 0.00000,C 180.00000} ; insert
  LIN {X -15854.028,Y -1023.446,Z -406.648,A -89.93308,B 0.00000,C 180.00000} ; release
  LIN {X -15854.028,Y -1023.446,Z -106.648,A -89.93308,B 0.00000,C 180.00000} ; retreat
  ; Step 66, bar 3281
  LIN {X -15704.028,Y -1023.446,Z 793.100,A -89.93308,B 0.00000,C 180.00000} ; outside
  LIN {X -15704.028,Y -1023.446,Z -156.648,A -89.93308,B 0.00000,C 180.00000} ; preinsert
  LIN {X -15704.028,Y -1023.446,Z -406.648,A -89.93308,B 0.00000,C 180.00000} ; insert
  LIN {X -15704.028,Y -1023.446,Z -406.648,A -89.93308,B 0.00000,C 180.00000} ; release
  LIN {X -15704.028,Y -1023.446,Z -106.648,A -89.93308,B 0.00000,C 180.00000} ; retreat
  ; Step 67, bar 3361
  LIN {X 15704.060,Y -1023.446,Z 793.100,A -89.99904,B 0.00000,C 180.00000} ; outside
  LIN {X 15704.060,Y -1023.446,Z -156.648,A -89.99904,B 0.00000,C 180.00000} ; preinsert
  LIN {X 15704.060,Y -1023.446,Z -406.648,A -89.99904,B 0.00000,C 180.00000} ; insert
  LIN {X 15704.060,Y -1023.446,Z -406.648,A -89.99904,B 0.00000,C 180.00000} ; release
  LIN {X 15704.060,Y -1023.446,Z -106.648,A -89.99904,B 0.00000,C 180.00000} ; retreat
  ; Step 68, bar 3363
  LIN {X 15854.060,Y -1023.446,Z 793.100,A -89.99904,B 0.00000,C 180.00000} ; outside
  LIN {X 15854.060,Y -1023.446,Z -156.648,A -89.99904,B 0.00000,C 180.00000} ; preinsert
  LIN {X 15854.060,Y -1023.446,Z -406.648,A -89.99904,B 0.00000,C 180.00000} ; insert
  LIN {X 15854.060,Y -1023.446,Z -406.648,A -89.99904,B 0.00000,C 180.00000} ; release
  LIN {X 15854.060,Y -1023.446,Z -106.648,A -89.99904,B 0.00000,C 180.00000} ; retreat
  ; Step 69, bar 3323
  LIN {X -15854.060,Y 1023.446,Z 793.100,A 90.00096,B 0.00000,C 180.00000} ; outside
  LIN {X -15854.060,Y 1023.446,Z -156.648,A 90.00096,B 0.00000,C 180.00000} ; preinsert
  LIN {X -15854.060,Y 1023.446,Z -406.648,A 90.00096,B 0.00000,C 180.00000} ; insert
  LIN {X -15854.060,Y 1023.446,Z -406.648,A 90.00096,B 0.00000,C 180.00000} ; release
  LIN {X -15854.060,Y 1023.446,Z -106.648,A 90.00096,B 0.00000,C 180.00000} ; retreat
  ; Step 70, bar 3321
  LIN {X -15704.060,Y 1023.446,Z 793.100,A 90.00096,B 0.00000,C 180.00000} ; outside
  LIN {X -15704.060,Y 1023.446,Z -156.648,A 90.00096,B 0.00000,C 180.00000} ; preinsert
  LIN {X -15704.060,Y 1023.446,Z -406.648,A 90.00096,B 0.00000,C 180.00000} ; insert
  LIN {X -15704.060,Y 1023.446,Z -406.648,A 90.00096,B 0.00000,C 180.00000} ; release
  LIN {X -15704.060,Y 1023.446,Z -106.648,A 90.00096,B 0.00000,C 180.00000} ; retreat
  ; Step 71, bar 3401
  LIN {X 15704.028,Y 1023.446,Z 793.100,A 90.06692,B 0.00000,C 180.00000} ; outside
  LIN {X 15704.028,Y 1023.446,Z -156.648,A 90.06692,B 0.00000,C 180.00000} ; preinsert
  LIN {X 15704.028,Y 1023.446,Z -406.648,A 90.06692,B 0.00000,C 180.00000} ; insert
  LIN {X 15704.028,Y 1023.446,Z -406.648,A 90.06692,B 0.00000,C 180.00000} ; release
  LIN {X 15704.028,Y 1023.446,Z -106.648,A 90.06692,B 0.00000,C 180.00000} ; retreat
  ; Step 72, bar 3403
  LIN {X 15854.028,Y 1023.446,Z 793.100,A 90.06692,B 0.00000,C 180.00000} ; outside
  LIN {X 15854.028,Y 1023.446,Z -156.648,A 90.06692,B 0.00000,C 180.00000} ; preinsert
  LIN {X 15854.028,Y 1023.446,Z -406.648,A 90.06692,B 0.00000,C 180.00000} ; insert
  LIN {X 15854.028,Y 1023.446,Z -406.648,A 90.06692,B 0.00000,C 180.00000} ; release
  LIN {X 15854.028,Y 1023.446,Z -106.648,A 90.06692,B 0.00000,C 180.00000} ; retreat
  ; Step 73, bar 3280
  LIN {X -15629.028,Y -1023.446,Z 793.100,A -89.93308,B 0.00000,C 180.00000} ; outside
  LIN {X -15629.028,Y -1023.446,Z -156.648,A -89.93308,B 0.00000,C 180.00000} ; preinsert
  LIN {X -15629.028,Y -1023.446,Z -406.648,A -89.93308,B 0.00000,C 180.00000} ; insert
  LIN {X -15629.028,Y -1023.446,Z -406.648,A -89.93308,B 0.00000,C 180.00000} ; release
  LIN {X -15629.028,Y -1023.446,Z -106.648,A -89.93308,B 0.00000,C 180.00000} ; retreat
  ; Step 74, bar 3277
  LIN {X -15470.940,Y -1023.446,Z 793.100,A -89.99904,B 0.00000,C 180.00000} ; outside
  LIN {X -15470.940,Y -1023.446,Z -156.648,A -89.99904,B 0.00000,C 180.00000} ; preinsert
  LIN {X -15470.940,Y -1023.446,Z -406.648,A -89.99904,B 0.00000,C 180.00000} ; insert
  LIN {X -15470.940,Y -1023.446,Z -406.648,A -89.99904,B 0.00000,C 180.00000} ; release
  LIN {X -15470.940,Y -1023.446,Z -106.648,A -89.99904,B 0.00000,C 180.00000} ; retreat
  ; Step 75, bar 3357
  LIN {X 15470.972,Y -1023.446,Z 793.100,A -89.93308,B 0.00000,C 180.00000} ; outside
  LIN {X 15470.972,Y -1023.446,Z -156.648,A -89.93308,B 0.00000,C 180.00000} ; preinsert
  LIN {X 15470.972,Y -1023.446,Z -406.648,A -89.93308,B 0.00000,C 180.00000} ; insert
  LIN {X 15470.972,Y -1023.446,Z -406.648,A -89.93308,B 0.00000,C 180.00000} ; release
  LIN {X 15470.972,Y -1023.446,Z -106.648,A -89.93308,B 0.00000,C 180.00000} ; retreat
  ; Step 76, bar 3360
  LIN {X 15629.060,Y -1023.446,Z 793.100,A -89.99904,B 0.00000,C 180.00000} ; outside
  LIN {X 15629.060,Y -1023.446,Z -156.648,A -89.99904,B 0.00000,C 180.00000} ; preinsert
  LIN {X 15629.060,Y -1023.446,Z -406.648,A -89.99904,B 0.00000,C 180.00000} ; insert
  LIN {X 15629.060,Y -1023.446,Z -406.648,A -89.99904,B 0.00000,C 180.00000} ; release
  LIN {X 15629.060,Y -1023.446,Z -106.648,A -89.99904,B 0.00000,C 180.00000} ; retreat
  ; Step 77, bar 3320
  LIN {X -15629.060,Y 1023.446,Z 793.100,A 90.00096,B 0.00000,C 180.00000} ; outside
  LIN {X -15629.060,Y 1023.446,Z -156.648,A 90.00096,B 0.00000,C 180.00000} ; preinsert
  LIN {X -15629.060,Y 1023.446,Z -406.648,A 90.00096,B 0.00000,C 180.00000} ; insert
  LIN {X -15629.060,Y 1023.446,Z -406.648,A 90.00096,B 0.00000,C 180.00000} ; release
  LIN {X -15629.060,Y 1023.446,Z -106.648,A 90.00096,B 0.00000,C 180.00000} ; retreat
  ; Step 78, bar 3317
  LIN {X -15470.972,Y 1023.446,Z 793.100,A 90.06692,B 0.00000,C 180.00000} ; outside
  LIN {X -15470.972,Y 1023.446,Z -156.648,A 90.06692,B 0.00000,C 180.00000} ; preinsert
  LIN {X -15470.972,Y 1023.446,Z -406.648,A 90.06692,B 0.00000,C 180.00000} ; insert
  LIN {X -15470.972,Y 1023.446,Z -406.648,A 90.06692,B 0.00000,C 180.00000} ; release
  LIN {X -15470.972,Y 1023.446,Z -106.648,A 90.06692,B 0.00000,C 180.00000} ; retreat
  ; Step 79, bar 3397
  LIN {X 15470.940,Y 1023.446,Z 793.100,A 90.00096,B 0.00000,C 180.00000} ; outside
  LIN {X 15470.940,Y 1023.446,Z -156.648,A 90.00096,B 0.00000,C 180.00000} ; preinsert
  LIN {X 15470.940,Y 1023.446,Z -406.648,A 90.00096,B 0.00000,C 180.00000} ; insert
  LIN {X 15470.940,Y 1023.446,Z -406.648,A 90.00096,B 0.00000,C 180.00000} ; release
  LIN {X 15470.940,Y 1023.446,Z -106.648,A 90.00096,B 0.00000,C 180.00000} ; retreat
  ; Step 80, bar 3400
  LIN {X 15629.028,Y 1023.446,Z 793.100,A 90.06692,B 0.00000,C 180.00000} ; outside
  LIN {X 15629.028,Y 1023.446,Z -156.648,A 90.06692,B 0.00000,C 180.00000} ; preinsert
  LIN {X 15629.028,Y 1023.446,Z -406.648,A 90.06692,B 0.00000,C 180.00000} ; insert
  LIN {X 15629.028,Y 1023.446,Z -406.648,A 90.06692,B 0.00000,C 180.00000} ; release
  LIN {X 15629.028,Y 1023.446,Z -106.648,A 90.06692,B 0.00000,C 180.00000} ; retreat
  ; Step 81, bar 3262
  LIN {X -14779.028,Y -1023.446,Z 793.100,A -89.93308,B 0.00000,C 180.00000} ; outside
  LIN {X -14779.028,Y -1023.446,Z -156.648,A -89.93308,B 0.00000,C 180.00000} ; preinsert
  LIN {X -14779.028,Y -1023.446,Z -406.648,A -89.93308,B 0.00000,C 180.00000} ; insert
  LIN {X -14779.028,Y -1023.446,Z -406.648,A -89.93308,B 0.00000,C 180.00000} ; release
  LIN {X -14779.028,Y -1023.446,Z -106.648,A -89.93308,B 0.00000,C 180.00000} ; retreat
  ; Step 82, bar 3258
  LIN {X -14395.940,Y -1023.446,Z 793.100,A -89.99904,B 0.00000,C 180.00000} ; outside
  LIN {X -14395.940,Y -1023.446,Z -156.648,A -89.99904,B 0.00000,C 180.00000} ; preinsert
  LIN {X -14395.940,Y -1023.446,Z -406.648,A -89.99904,B 0.00000,C 180.00000} ; insert
  LIN {X -14395.940,Y -1023.446,Z -406.648,A -89.99904,B 0.00000,C 180.00000} ; release
  LIN {X -14395.940,Y -1023.446,Z -106.648,A -89.99904,B 0.00000,C 180.00000} ; retreat
  ; Step 83, bar 3259
  LIN {X -14320.940,Y -1023.446,Z 793.100,A -89.99904,B 0.00000,C 180.00000} ; outside
  LIN {X -14320.940,Y -1023.446,Z -156.648,A -89.99904,B 0.00000,C 180.00000} ; preinsert
  LIN {X -14320.940,Y -1023.446,Z -406.648,A -89.99904,B 0.00000,C 180.00000} ; insert
  LIN {X -14320.940,Y -1023.446,Z -406.648,A -89.99904,B 0.00000,C 180.00000} ; release
  LIN {X -14320.940,Y -1023.446,Z -106.648,A -89.99904,B 0.00000,C 180.00000} ; retreat
  ; Step 84, bar 3339
  LIN {X 14320.972,Y -1023.446,Z 793.100,A -89.93308,B 0.00000,C 180.00000} ; outside
  LIN {X 14320.972,Y -1023.446,Z -156.648,A -89.93308,B 0.00000,C 180.00000} ; preinsert
  LIN {X 14320.972,Y -1023.446,Z -406.648,A -89.93308,B 0.00000,C 180.00000} ; insert
  LIN {X 14320.972,Y -1023.446,Z -406.648,A -89.93308,B 0.00000,C 180.00000} ; release
  LIN {X 14320.972,Y -1023.446,Z -106.648,A -89.93308,B 0.00000,C 180.00000} ; retreat
  ; Step 85, bar 3338
  LIN {X 14395.972,Y -1023.446,Z 793.100,A -89.93308,B 0.00000,C 180.00000} ; outside
  LIN {X 14395.972,Y -1023.446,Z -156.648,A -89.93308,B 0.00000,C 180.00000} ; preinsert
  LIN {X 14395.972,Y -1023.446,Z -406.648,A -89.93308,B 0.00000,C 180.00000} ; insert
  LIN {X 14395.972,Y -1023.446,Z -406.648,A -89.93308,B 0.00000,C 180.00000} ; release
  LIN {X 14395.972,Y -1023.446,Z -106.648,A -89.93308,B 0.00000,C 180.00000} ; retreat
  ; Step 86, bar 3342
  LIN {X 14779.060,Y -1023.446,Z 793.100,A -89.99904,B 0.00000,C 180.00000} ; outside
  LIN {X 14779.060,Y -1023.446,Z -156.648,A -89.99904,B 0.00000,C 180.00000} ; preinsert
  LIN {X 14779.060,Y -1023.446,Z -406.648,A -89.99904,B 0.00000,C 180.00000} ; insert
  LIN {X 14779.060,Y -1023.446,Z -406.648,A -89.99904,B 0.00000,C 180.00000} ; release
  LIN {X 14779.060,Y -1023.446,Z -106.648,A -89.99904,B 0.00000,C 180.00000} ; retreat
  ; Step 87, bar 3302
  LIN {X -14779.060,Y 1023.446,Z 793.100,A 90.00096,B 0.00000,C 180.00000} ; outside
  LIN {X -14779.060,Y 1023.446,Z -156.648,A 90.00096,B 0.00000,C 180.00000} ; preinsert
  LIN {X -14779.060,Y 1023.446,Z -406.648,A 90.00096,B 0.00000,C 180.00000} ; insert
  LIN {X -14779.060,Y 1023.446,Z -406.648,A 90.00096,B 0.00000,C 180.00000} ; release
  LIN {X -14779.060,Y 1023.446,Z -106.648,A 90.00096,B 0.00000,C 180.00000} ; retreat
  ; Step 88, bar 3298
  LIN {X -14395.972,Y 1023.446,Z 793.100,A 90.06692,B 0.00000,C 180.00000} ; outside
  LIN {X -14395.972,Y 1023.446,Z -156.648,A 90.06692,B 0.00000,C 180.00000} ; preinsert
  LIN {X -14395.972,Y 1023.446,Z -406.648,A 90.06692,B 0.00000,C 180.00000} ; insert
  LIN {X -14395.972,Y 1023.446,Z -406.648,A 90.06692,B 0.00000,C 180.00000} ; release
  LIN {X -14395.972,Y 1023.446,Z -106.648,A 90.06692,B 0.00000,C 180.00000} ; retreat
  ; Step 89, bar 3299
  LIN {X -14320.972,Y 1023.446,Z 793.100,A 90.06692,B 0.00000,C 180.00000} ; outside
  LIN {X -14320.972,Y 1023.446,Z -156.648,A 90.06692,B 0.00000,C 180.00000} ; preinsert
  LIN {X -14320.972,Y 1023.446,Z -406.648,A 90.06692,B 0.00000,C 180.00000} ; insert
  LIN {X -14320.972,Y 1023.446,Z -406.648,A 90.06692,B 0.00000,C 180.00000} ; release
  LIN {X -14320.972,Y 1023.446,Z -106.648,A 90.06692,B 0.00000,C 180.00000} ; retreat
  ; Step 90, bar 3379
  LIN {X 14320.940,Y 1023.446,Z 793.100,A 90.00096,B 0.00000,C 180.00000} ; outside
  LIN {X 14320.940,Y 1023.446,Z -156.648,A 90.00096,B 0.00000,C 180.00000} ; preinsert
  LIN {X 14320.940,Y 1023.446,Z -406.648,A 90.00096,B 0.00000,C 180.00000} ; insert
  LIN {X 14320.940,Y 1023.446,Z -406.648,A 90.00096,B 0.00000,C 180.00000} ; release
  LIN {X 14320.940,Y 1023.446,Z -106.648,A 90.00096,B 0.00000,C 180.00000} ; retreat
  ; Step 91, bar 3378
  LIN {X 14395.940,Y 1023.446,Z 793.100,A 90.00096,B 0.00000,C 180.00000} ; outside
  LIN {X 14395.940,Y 1023.446,Z -156.648,A 90.00096,B 0.00000,C 180.00000} ; preinsert
  LIN {X 14395.940,Y 1023.446,Z -406.648,A 90.00096,B 0.00000,C 180.00000} ; insert
  LIN {X 14395.940,Y 1023.446,Z -406.648,A 90.00096,B 0.00000,C 180.00000} ; release
  LIN {X 14395.940,Y 1023.446,Z -106.648,A 90.00096,B 0.00000,C 180.00000} ; retreat
  ; Step 92, bar 3382
  LIN {X 14779.028,Y 1023.446,Z 793.100,A 90.06692,B 0.00000,C 180.00000} ; outside
  LIN {X 14779.028,Y 1023.446,Z -156.648,A 90.06692,B 0.00000,C 180.00000} ; preinsert
  LIN {X 14779.028,Y 1023.446,Z -406.648,A 90.06692,B 0.00000,C 180.00000} ; insert
  LIN {X 14779.028,Y 1023.446,Z -406.648,A 90.06692,B 0.00000,C 180.00000} ; release
  LIN {X 14779.028,Y 1023.446,Z -106.648,A 90.06692,B 0.00000,C 180.00000} ; retreat
  ; Step 93, bar 3263
  LIN {X -14854.028,Y -1023.446,Z 793.100,A -89.93308,B 0.00000,C 180.00000} ; outside
  LIN {X -14854.028,Y -1023.446,Z -156.648,A -89.93308,B 0.00000,C 180.00000} ; preinsert
  LIN {X -14854.028,Y -1023.446,Z -406.648,A -89.93308,B 0.00000,C 180.00000} ; insert
  LIN {X -14854.028,Y -1023.446,Z -406.648,A -89.93308,B 0.00000,C 180.00000} ; release
  LIN {X -14854.028,Y -1023.446,Z -106.648,A -89.93308,B 0.00000,C 180.00000} ; retreat
  ; Step 94, bar 3261
  LIN {X -14704.028,Y -1023.446,Z 793.100,A -89.93308,B 0.00000,C 180.00000} ; outside
  LIN {X -14704.028,Y -1023.446,Z -156.648,A -89.93308,B 0.00000,C 180.00000} ; preinsert
  LIN {X -14704.028,Y -1023.446,Z -406.648,A -89.93308,B 0.00000,C 180.00000} ; insert
  LIN {X -14704.028,Y -1023.446,Z -406.648,A -89.93308,B 0.00000,C 180.00000} ; release
  LIN {X -14704.028,Y -1023.446,Z -106.648,A -89.93308,B 0.00000,C 180.00000} ; retreat
  ; Step 95, bar 3341
  LIN {X 14704.060,Y -1023.446,Z 793.100,A -89.99904,B 0.00000,C 180.00000} ; outside
  LIN {X 14704.060,Y -1023.446,Z -156.648,A -89.99904,B 0.00000,C 180.00000} ; preinsert
  LIN {X 14704.060,Y -1023.446,Z -406.648,A -89.99904,B 0.00000,C 180.00000} ; insert
  LIN {X 14704.060,Y -1023.446,Z -406.648,A -89.99904,B 0.00000,C 180.00000} ; release
  LIN {X 14704.060,Y -1023.446,Z -106.648,A -89.99904,B 0.00000,C 180.00000} ; retreat
  ; Step 96, bar 3343
  LIN {X 14854.060,Y -1023.446,Z 793.100,A -89.99904,B 0.00000,C 180.00000} ; outside
  LIN {X 14854.060,Y -1023.446,Z -156.648,A -89.99904,B 0.00000,C 180.00000} ; preinsert
  LIN {X 14854.060,Y -1023.446,Z -406.648,A -89.99904,B 0.00000,C 180.00000} ; insert
  LIN {X 14854.060,Y -1023.446,Z -406.648,A -89.99904,B 0.00000,C 180.00000} ; release
  LIN {X 14854.060,Y -1023.446,Z -106.648,A -89.99904,B 0.00000,C 180.00000} ; retreat
  ; Step 97, bar 3303
  LIN {X -14854.060,Y 1023.446,Z 793.100,A 90.00096,B 0.00000,C 180.00000} ; outside
  LIN {X -14854.060,Y 1023.446,Z -156.648,A 90.00096,B 0.00000,C 180.00000} ; preinsert
  LIN {X -14854.060,Y 1023.446,Z -406.648,A 90.00096,B 0.00000,C 180.00000} ; insert
  LIN {X -14854.060,Y 1023.446,Z -406.648,A 90.00096,B 0.00000,C 180.00000} ; release
  LIN {X -14854.060,Y 1023.446,Z -106.648,A 90.00096,B 0.00000,C 180.00000} ; retreat
  ; Step 98, bar 3301
  LIN {X -14704.060,Y 1023.446,Z 793.100,A 90.00096,B 0.00000,C 180.00000} ; outside
  LIN {X -14704.060,Y 1023.446,Z -156.648,A 90.00096,B 0.00000,C 180.00000} ; preinsert
  LIN {X -14704.060,Y 1023.446,Z -406.648,A 90.00096,B 0.00000,C 180.00000} ; insert
  LIN {X -14704.060,Y 1023.446,Z -406.648,A 90.00096,B 0.00000,C 180.00000} ; release
  LIN {X -14704.060,Y 1023.446,Z -106.648,A 90.00096,B 0.00000,C 180.00000} ; retreat
  ; Step 99, bar 3381
  LIN {X 14704.028,Y 1023.446,Z 793.100,A 90.06692,B 0.00000,C 180.00000} ; outside
  LIN {X 14704.028,Y 1023.446,Z -156.648,A 90.06692,B 0.00000,C 180.00000} ; preinsert
  LIN {X 14704.028,Y 1023.446,Z -406.648,A 90.06692,B 0.00000,C 180.00000} ; insert
  LIN {X 14704.028,Y 1023.446,Z -406.648,A 90.06692,B 0.00000,C 180.00000} ; release
  LIN {X 14704.028,Y 1023.446,Z -106.648,A 90.06692,B 0.00000,C 180.00000} ; retreat
  ; Step 100, bar 3383
  LIN {X 14854.028,Y 1023.446,Z 793.100,A 90.06692,B 0.00000,C 180.00000} ; outside
  LIN {X 14854.028,Y 1023.446,Z -156.648,A 90.06692,B 0.00000,C 180.00000} ; preinsert
  LIN {X 14854.028,Y 1023.446,Z -406.648,A 90.06692,B 0.00000,C 180.00000} ; insert
  LIN {X 14854.028,Y 1023.446,Z -406.648,A 90.06692,B 0.00000,C 180.00000} ; release
  LIN {X 14854.028,Y 1023.446,Z -106.648,A 90.06692,B 0.00000,C 180.00000} ; retreat
  ; Step 101, bar 3260
  LIN {X -14629.028,Y -1023.446,Z 793.100,A -89.93308,B 0.00000,C 180.00000} ; outside
  LIN {X -14629.028,Y -1023.446,Z -156.648,A -89.93308,B 0.00000,C 180.00000} ; preinsert
  LIN {X -14629.028,Y -1023.446,Z -406.648,A -89.93308,B 0.00000,C 180.00000} ; insert
  LIN {X -14629.028,Y -1023.446,Z -406.648,A -89.93308,B 0.00000,C 180.00000} ; release
  LIN {X -14629.028,Y -1023.446,Z -106.648,A -89.93308,B 0.00000,C 180.00000} ; retreat
  ; Step 102, bar 3257
  LIN {X -14470.940,Y -1023.446,Z 793.100,A -89.99904,B 0.00000,C 180.00000} ; outside
  LIN {X -14470.940,Y -1023.446,Z -156.648,A -89.99904,B 0.00000,C 180.00000} ; preinsert
  LIN {X -14470.940,Y -1023.446,Z -406.648,A -89.99904,B 0.00000,C 180.00000} ; insert
  LIN {X -14470.940,Y -1023.446,Z -406.648,A -89.99904,B 0.00000,C 180.00000} ; release
  LIN {X -14470.940,Y -1023.446,Z -106.648,A -89.99904,B 0.00000,C 180.00000} ; retreat
  ; Step 103, bar 3337
  LIN {X 14470.972,Y -1023.446,Z 793.100,A -89.93308,B 0.00000,C 180.00000} ; outside
  LIN {X 14470.972,Y -1023.446,Z -156.648,A -89.93308,B 0.00000,C 180.00000} ; preinsert
  LIN {X 14470.972,Y -1023.446,Z -406.648,A -89.93308,B 0.00000,C 180.00000} ; insert
  LIN {X 14470.972,Y -1023.446,Z -406.648,A -89.93308,B 0.00000,C 180.00000} ; release
  LIN {X 14470.972,Y -1023.446,Z -106.648,A -89.93308,B 0.00000,C 180.00000} ; retreat
  ; Step 104, bar 3340
  LIN {X 14629.060,Y -1023.446,Z 793.100,A -89.99904,B 0.00000,C 180.00000} ; outside
  LIN {X 14629.060,Y -1023.446,Z -156.648,A -89.99904,B 0.00000,C 180.00000} ; preinsert
  LIN {X 14629.060,Y -1023.446,Z -406.648,A -89.99904,B 0.00000,C 180.00000} ; insert
  LIN {X 14629.060,Y -1023.446,Z -406.648,A -89.99904,B 0.00000,C 180.00000} ; release
  LIN {X 14629.060,Y -1023.446,Z -106.648,A -89.99904,B 0.00000,C 180.00000} ; retreat
  ; Step 105, bar 3300
  LIN {X -14629.060,Y 1023.446,Z 793.100,A 90.00096,B 0.00000,C 180.00000} ; outside
  LIN {X -14629.060,Y 1023.446,Z -156.648,A 90.00096,B 0.00000,C 180.00000} ; preinsert
  LIN {X -14629.060,Y 1023.446,Z -406.648,A 90.00096,B 0.00000,C 180.00000} ; insert
  LIN {X -14629.060,Y 1023.446,Z -406.648,A 90.00096,B 0.00000,C 180.00000} ; release
  LIN {X -14629.060,Y 1023.446,Z -106.648,A 90.00096,B 0.00000,C 180.00000} ; retreat
  ; Step 106, bar 3297
  LIN {X -14470.972,Y 1023.446,Z 793.100,A 90.06692,B 0.00000,C 180.00000} ; outside
  LIN {X -14470.972,Y 1023.446,Z -156.648,A 90.06692,B 0.00000,C 180.00000} ; preinsert
  LIN {X -14470.972,Y 1023.446,Z -406.648,A 90.06692,B 0.00000,C 180.00000} ; insert
  LIN {X -14470.972,Y 1023.446,Z -406.648,A 90.06692,B 0.00000,C 180.00000} ; release
  LIN {X -14470.972,Y 1023.446,Z -106.648,A 90.06692,B 0.00000,C 180.00000} ; retreat
  ; Step 107, bar 3377
  LIN {X 14470.940,Y 1023.446,Z 793.100,A 90.00096,B 0.00000,C 180.00000} ; outside
  LIN {X 14470.940,Y 1023.446,Z -156.648,A 90.00096,B 0.00000,C 180.00000} ; preinsert
  LIN {X 14470.940,Y 1023.446,Z -406.648,A 90.00096,B 0.00000,C 180.00000} ; insert
  LIN {X 14470.940,Y 1023.446,Z -406.648,A 90.00096,B 0.00000,C 180.00000} ; release
  LIN {X 14470.940,Y 1023.446,Z -106.648,A 90.00096,B 0.00000,C 180.00000} ; retreat
  ; Step 108, bar 3380
  LIN {X 14629.028,Y 1023.446,Z 793.100,A 90.06692,B 0.00000,C 180.00000} ; outside
  LIN {X 14629.028,Y 1023.446,Z -156.648,A 90.06692,B 0.00000,C 180.00000} ; preinsert
  LIN {X 14629.028,Y 1023.446,Z -406.648,A 90.06692,B 0.00000,C 180.00000} ; insert
  LIN {X 14629.028,Y 1023.446,Z -406.648,A 90.06692,B 0.00000,C 180.00000} ; release
  LIN {X 14629.028,Y 1023.446,Z -106.648,A 90.06692,B 0.00000,C 180.00000} ; retreat
  ; Step 109, bar 1862
  LIN {X 0.000,Y -2324.855,Z 792.630,A 0.00000,B 0.00000,C 180.00000} ; outside
  LIN {X 0.000,Y -2324.855,Z -84.730,A 0.00000,B 0.00000,C 180.00000} ; preinsert
  LIN {X 0.000,Y -2324.855,Z -334.730,A 0.00000,B 0.00000,C 180.00000} ; insert
  LIN {X 0.000,Y -2324.855,Z -334.730,A 0.00000,B 0.00000,C 180.00000} ; release
  LIN {X 0.000,Y -2324.855,Z -34.730,A 0.00000,B 0.00000,C 180.00000} ; retreat
  ; Step 110, bar 1875
  LIN {X 0.000,Y 2324.855,Z 792.630,A 0.00000,B 0.00000,C 180.00000} ; outside
  LIN {X 0.000,Y 2324.855,Z -84.730,A 0.00000,B 0.00000,C 180.00000} ; preinsert
  LIN {X 0.000,Y 2324.855,Z -334.730,A 0.00000,B 0.00000,C 180.00000} ; insert
  LIN {X 0.000,Y 2324.855,Z -334.730,A 0.00000,B 0.00000,C 180.00000} ; release
  LIN {X 0.000,Y 2324.855,Z -34.730,A 0.00000,B 0.00000,C 180.00000} ; retreat
  ; Step 111, bar 1863
  LIN {X 0.000,Y -2454.855,Z 792.630,A 0.00000,B 0.00000,C 180.00000} ; outside
  LIN {X 0.000,Y -2454.855,Z -69.788,A 0.00000,B 0.00000,C 180.00000} ; preinsert
  LIN {X 0.000,Y -2454.855,Z -319.788,A 0.00000,B 0.00000,C 180.00000} ; insert
  LIN {X 0.000,Y -2454.855,Z -319.788,A 0.00000,B 0.00000,C 180.00000} ; release
  LIN {X 0.000,Y -2454.855,Z -19.788,A 0.00000,B 0.00000,C 180.00000} ; retreat
  ; Step 112, bar 1876
  LIN {X 0.000,Y 2454.855,Z 792.630,A 0.00000,B 0.00000,C 180.00000} ; outside
  LIN {X 0.000,Y 2454.855,Z -69.788,A 0.00000,B 0.00000,C 180.00000} ; preinsert
  LIN {X 0.000,Y 2454.855,Z -319.788,A 0.00000,B 0.00000,C 180.00000} ; insert
  LIN {X 0.000,Y 2454.855,Z -319.788,A 0.00000,B 0.00000,C 180.00000} ; release
  LIN {X 0.000,Y 2454.855,Z -19.788,A 0.00000,B 0.00000,C 180.00000} ; retreat
  ; Step 113, bar 3287
  LIN {X -15736.114,Y -1213.921,Z 793.666,A 0.00932,B 0.00000,C 180.00000} ; outside
  LIN {X -15736.114,Y -1213.921,Z -168.174,A 0.00932,B 0.00000,C 180.00000} ; preinsert
  LIN {X -15736.114,Y -1213.921,Z -418.174,A 0.00932,B 0.00000,C 180.00000} ; insert
  LIN {X -15736.114,Y -1213.921,Z -418.174,A 0.00932,B 0.00000,C 180.00000} ; release
  LIN {X -15736.114,Y -1213.921,Z -118.174,A 0.00932,B 0.00000,C 180.00000} ; retreat
  ; Step 114, bar 3367
  LIN {X 15736.114,Y -1213.921,Z 793.666,A 179.99068,B 0.00000,C -180.00000} ; outside
  LIN {X 15736.114,Y -1213.921,Z -168.174,A 179.99068,B 0.00000,C -180.00000} ; preinsert
  LIN {X 15736.114,Y -1213.921,Z -418.174,A 179.99068,B 0.00000,C -180.00000} ; insert
  LIN {X 15736.114,Y -1213.921,Z -418.174,A 179.99068,B 0.00000,C -180.00000} ; release
  LIN {X 15736.114,Y -1213.921,Z -118.174,A 179.99068,B 0.00000,C -180.00000} ; retreat
  ; Step 115, bar 3276
  LIN {X -15736.114,Y -1128.921,Z 793.666,A 0.00932,B 0.00000,C 180.00000} ; outside
  LIN {X -15736.114,Y -1128.921,Z -168.174,A 0.00932,B 0.00000,C 180.00000} ; preinsert
  LIN {X -15736.114,Y -1128.921,Z -418.174,A 0.00932,B 0.00000,C 180.00000} ; insert
  LIN {X -15736.114,Y -1128.921,Z -418.174,A 0.00932,B 0.00000,C 180.00000} ; release
  LIN {X -15736.114,Y -1128.921,Z -118.174,A 0.00932,B 0.00000,C 180.00000} ; retreat
  ; Step 116, bar 3356
  LIN {X 15736.114,Y -1128.921,Z 793.666,A 179.99068,B 0.00000,C -180.00000} ; outside
  LIN {X 15736.114,Y -1128.921,Z -168.174,A 179.99068,B 0.00000,C -180.00000} ; preinsert
  LIN {X 15736.114,Y -1128.921,Z -418.174,A 179.99068,B 0.00000,C -180.00000} ; insert
  LIN {X 15736.114,Y -1128.921,Z -418.174,A 179.99068,B 0.00000,C -180.00000} ; release
  LIN {X 15736.114,Y -1128.921,Z -118.174,A 179.99068,B 0.00000,C -180.00000} ; retreat
  ; Step 117, bar 3284
  LIN {X -15736.114,Y -970.921,Z 793.666,A 0.00932,B 0.00000,C 180.00000} ; outside
  LIN {X -15736.114,Y -970.921,Z -168.174,A 0.00932,B 0.00000,C 180.00000} ; preinsert
  LIN {X -15736.114,Y -970.921,Z -418.174,A 0.00932,B 0.00000,C 180.00000} ; insert
  LIN {X -15736.114,Y -970.921,Z -418.174,A 0.00932,B 0.00000,C 180.00000} ; release
  LIN {X -15736.114,Y -970.921,Z -118.174,A 0.00932,B 0.00000,C 180.00000} ; retreat
  ; Step 118, bar 3364
  LIN {X 15736.114,Y -970.921,Z 793.666,A 179.99068,B 0.00000,C 180.00000} ; outside
  LIN {X 15736.114,Y -970.921,Z -168.174,A 179.99068,B 0.00000,C 180.00000} ; preinsert
  LIN {X 15736.114,Y -970.921,Z -418.174,A 179.99068,B 0.00000,C 180.00000} ; insert
  LIN {X 15736.114,Y -970.921,Z -418.174,A 179.99068,B 0.00000,C 180.00000} ; release
  LIN {X 15736.114,Y -970.921,Z -118.174,A 179.99068,B 0.00000,C 180.00000} ; retreat
  ; Step 119, bar 3285
  LIN {X -15736.114,Y -885.921,Z 793.666,A 0.00932,B 0.00000,C 180.00000} ; outside
  LIN {X -15736.114,Y -885.921,Z -168.174,A 0.00932,B 0.00000,C 180.00000} ; preinsert
  LIN {X -15736.114,Y -885.921,Z -418.174,A 0.00932,B 0.00000,C 180.00000} ; insert
  LIN {X -15736.114,Y -885.921,Z -418.174,A 0.00932,B 0.00000,C 180.00000} ; release
  LIN {X -15736.114,Y -885.921,Z -118.174,A 0.00932,B 0.00000,C 180.00000} ; retreat
  ; Step 120, bar 3365
  LIN {X 15736.114,Y -885.921,Z 793.666,A 179.99068,B 0.00000,C 180.00000} ; outside
  LIN {X 15736.114,Y -885.921,Z -168.174,A 179.99068,B 0.00000,C 180.00000} ; preinsert
  LIN {X 15736.114,Y -885.921,Z -418.174,A 179.99068,B 0.00000,C 180.00000} ; insert
  LIN {X 15736.114,Y -885.921,Z -418.174,A 179.99068,B 0.00000,C 180.00000} ; release
  LIN {X 15736.114,Y -885.921,Z -118.174,A 179.99068,B 0.00000,C 180.00000} ; retreat
  ; Step 121, bar 3286
  LIN {X -15736.114,Y -800.921,Z 793.666,A 0.00932,B 0.00000,C 180.00000} ; outside
  LIN {X -15736.114,Y -800.921,Z -168.174,A 0.00932,B 0.00000,C 180.00000} ; preinsert
  LIN {X -15736.114,Y -800.921,Z -418.174,A 0.00932,B 0.00000,C 180.00000} ; insert
  LIN {X -15736.114,Y -800.921,Z -418.174,A 0.00932,B 0.00000,C 180.00000} ; release
  LIN {X -15736.114,Y -800.921,Z -118.174,A 0.00932,B 0.00000,C 180.00000} ; retreat
  ; Step 122, bar 3366
  LIN {X 15736.114,Y -800.921,Z 793.666,A 179.99068,B 0.00000,C 180.00000} ; outside
  LIN {X 15736.114,Y -800.921,Z -168.174,A 179.99068,B 0.00000,C 180.00000} ; preinsert
  LIN {X 15736.114,Y -800.921,Z -418.174,A 179.99068,B 0.00000,C 180.00000} ; insert
  LIN {X 15736.114,Y -800.921,Z -418.174,A 179.99068,B 0.00000,C 180.00000} ; release
  LIN {X 15736.114,Y -800.921,Z -118.174,A 179.99068,B 0.00000,C 180.00000} ; retreat
  ; Step 123, bar 3326
  LIN {X -15736.114,Y 800.921,Z 793.666,A -0.00932,B 0.00000,C 180.00000} ; outside
  LIN {X -15736.114,Y 800.921,Z -168.174,A -0.00932,B 0.00000,C 180.00000} ; preinsert
  LIN {X -15736.114,Y 800.921,Z -418.174,A -0.00932,B 0.00000,C 180.00000} ; insert
  LIN {X -15736.114,Y 800.921,Z -418.174,A -0.00932,B 0.00000,C 180.00000} ; release
  LIN {X -15736.114,Y 800.921,Z -118.174,A -0.00932,B 0.00000,C 180.00000} ; retreat
  ; Step 124, bar 3406
  LIN {X 15736.114,Y 800.921,Z 793.666,A -179.99068,B 0.00000,C -180.00000} ; outside
  LIN {X 15736.114,Y 800.921,Z -168.174,A -179.99068,B 0.00000,C -180.00000} ; preinsert
  LIN {X 15736.114,Y 800.921,Z -418.174,A -179.99068,B 0.00000,C -180.00000} ; insert
  LIN {X 15736.114,Y 800.921,Z -418.174,A -179.99068,B 0.00000,C -180.00000} ; release
  LIN {X 15736.114,Y 800.921,Z -118.174,A -179.99068,B 0.00000,C -180.00000} ; retreat
  ; Step 125, bar 3325
  LIN {X -15736.114,Y 885.921,Z 793.666,A -0.00932,B 0.00000,C 180.00000} ; outside
  LIN {X -15736.114,Y 885.921,Z -168.174,A -0.00932,B 0.00000,C 180.00000} ; preinsert
  LIN {X -15736.114,Y 885.921,Z -418.174,A -0.00932,B 0.00000,C 180.00000} ; insert
  LIN {X -15736.114,Y 885.921,Z -418.174,A -0.00932,B 0.00000,C 180.00000} ; release
  LIN {X -15736.114,Y 885.921,Z -118.174,A -0.00932,B 0.00000,C 180.00000} ; retreat
  ; Step 126, bar 3405
  LIN {X 15736.114,Y 885.921,Z 793.666,A -179.99068,B 0.00000,C -180.00000} ; outside
  LIN {X 15736.114,Y 885.921,Z -168.174,A -179.99068,B 0.00000,C -180.00000} ; preinsert
  LIN {X 15736.114,Y 885.921,Z -418.174,A -179.99068,B 0.00000,C -180.00000} ; insert
  LIN {X 15736.114,Y 885.921,Z -418.174,A -179.99068,B 0.00000,C -180.00000} ; release
  LIN {X 15736.114,Y 885.921,Z -118.174,A -179.99068,B 0.00000,C -180.00000} ; retreat
  ; Step 127, bar 3324
  LIN {X -15736.114,Y 970.921,Z 793.666,A -0.00932,B 0.00000,C 180.00000} ; outside
  LIN {X -15736.114,Y 970.921,Z -168.174,A -0.00932,B 0.00000,C 180.00000} ; preinsert
  LIN {X -15736.114,Y 970.921,Z -418.174,A -0.00932,B 0.00000,C 180.00000} ; insert
  LIN {X -15736.114,Y 970.921,Z -418.174,A -0.00932,B 0.00000,C 180.00000} ; release
  LIN {X -15736.114,Y 970.921,Z -118.174,A -0.00932,B 0.00000,C 180.00000} ; retreat
  ; Step 128, bar 3404
  LIN {X 15736.114,Y 970.921,Z 793.666,A -179.99068,B 0.00000,C -180.00000} ; outside
  LIN {X 15736.114,Y 970.921,Z -168.174,A -179.99068,B 0.00000,C -180.00000} ; preinsert
  LIN {X 15736.114,Y 970.921,Z -418.174,A -179.99068,B 0.00000,C -180.00000} ; insert
  LIN {X 15736.114,Y 970.921,Z -418.174,A -179.99068,B 0.00000,C -180.00000} ; release
  LIN {X 15736.114,Y 970.921,Z -118.174,A -179.99068,B 0.00000,C -180.00000} ; retreat
  ; Step 129, bar 3316
  LIN {X -15736.114,Y 1128.921,Z 793.666,A -0.00932,B 0.00000,C 180.00000} ; outside
  LIN {X -15736.114,Y 1128.921,Z -168.174,A -0.00932,B 0.00000,C 180.00000} ; preinsert
  LIN {X -15736.114,Y 1128.921,Z -418.174,A -0.00932,B 0.00000,C 180.00000} ; insert
  LIN {X -15736.114,Y 1128.921,Z -418.174,A -0.00932,B 0.00000,C 180.00000} ; release
  LIN {X -15736.114,Y 1128.921,Z -118.174,A -0.00932,B 0.00000,C 180.00000} ; retreat
  ; Step 130, bar 3396
  LIN {X 15736.114,Y 1128.921,Z 793.666,A -179.99068,B 0.00000,C -180.00000} ; outside
  LIN {X 15736.114,Y 1128.921,Z -168.174,A -179.99068,B 0.00000,C -180.00000} ; preinsert
  LIN {X 15736.114,Y 1128.921,Z -418.174,A -179.99068,B 0.00000,C -180.00000} ; insert
  LIN {X 15736.114,Y 1128.921,Z -418.174,A -179.99068,B 0.00000,C -180.00000} ; release
  LIN {X 15736.114,Y 1128.921,Z -118.174,A -179.99068,B 0.00000,C -180.00000} ; retreat
  ; Step 131, bar 3327
  LIN {X -15736.114,Y 1213.921,Z 793.666,A -0.00932,B 0.00000,C 180.00000} ; outside
  LIN {X -15736.114,Y 1213.921,Z -168.174,A -0.00932,B 0.00000,C 180.00000} ; preinsert
  LIN {X -15736.114,Y 1213.921,Z -418.174,A -0.00932,B 0.00000,C 180.00000} ; insert
  LIN {X -15736.114,Y 1213.921,Z -418.174,A -0.00932,B 0.00000,C 180.00000} ; release
  LIN {X -15736.114,Y 1213.921,Z -118.174,A -0.00932,B 0.00000,C 180.00000} ; retreat
  ; Step 132, bar 3407
  LIN {X 15736.114,Y 1213.921,Z 793.666,A -179.99068,B 0.00000,C -180.00000} ; outside
  LIN {X 15736.114,Y 1213.921,Z -168.174,A -179.99068,B 0.00000,C -180.00000} ; preinsert
  LIN {X 15736.114,Y 1213.921,Z -418.174,A -179.99068,B 0.00000,C -180.00000} ; insert
  LIN {X 15736.114,Y 1213.921,Z -418.174,A -179.99068,B 0.00000,C -180.00000} ; release
  LIN {X 15736.114,Y 1213.921,Z -118.174,A -179.99068,B 0.00000,C -180.00000} ; retreat
  ; Step 133, bar 3267
  LIN {X -14736.114,Y -1213.921,Z 793.666,A 0.00932,B 0.00000,C 180.00000} ; outside
  LIN {X -14736.114,Y -1213.921,Z -168.174,A 0.00932,B 0.00000,C 180.00000} ; preinsert
  LIN {X -14736.114,Y -1213.921,Z -418.174,A 0.00932,B 0.00000,C 180.00000} ; insert
  LIN {X -14736.114,Y -1213.921,Z -418.174,A 0.00932,B 0.00000,C 180.00000} ; release
  LIN {X -14736.114,Y -1213.921,Z -118.174,A 0.00932,B 0.00000,C 180.00000} ; retreat
  ; Step 134, bar 3347
  LIN {X 14736.114,Y -1213.921,Z 793.666,A 179.99068,B 0.00000,C -180.00000} ; outside
  LIN {X 14736.114,Y -1213.921,Z -168.174,A 179.99068,B 0.00000,C -180.00000} ; preinsert
  LIN {X 14736.114,Y -1213.921,Z -418.174,A 179.99068,B 0.00000,C -180.00000} ; insert
  LIN {X 14736.114,Y -1213.921,Z -418.174,A 179.99068,B 0.00000,C -180.00000} ; release
  LIN {X 14736.114,Y -1213.921,Z -118.174,A 179.99068,B 0.00000,C -180.00000} ; retreat
  ; Step 135, bar 3256
  LIN {X -14736.114,Y -1128.921,Z 793.666,A 0.00932,B 0.00000,C 180.00000} ; outside
  LIN {X -14736.114,Y -1128.921,Z -168.174,A 0.00932,B 0.00000,C 180.00000} ; preinsert
  LIN {X -14736.114,Y -1128.921,Z -418.174,A 0.00932,B 0.00000,C 180.00000} ; insert
  LIN {X -14736.114,Y -1128.921,Z -418.174,A 0.00932,B 0.00000,C 180.00000} ; release
  LIN {X -14736.114,Y -1128.921,Z -118.174,A 0.00932,B 0.00000,C 180.00000} ; retreat
  ; Step 136, bar 3336
  LIN {X 14736.114,Y -1128.921,Z 793.666,A 179.99068,B 0.00000,C -180.00000} ; outside
  LIN {X 14736.114,Y -1128.921,Z -168.174,A 179.99068,B 0.00000,C -180.00000} ; preinsert
  LIN {X 14736.114,Y -1128.921,Z -418.174,A 179.99068,B 0.00000,C -180.00000} ; insert
  LIN {X 14736.114,Y -1128.921,Z -418.174,A 179.99068,B 0.00000,C -180.00000} ; release
  LIN {X 14736.114,Y -1128.921,Z -118.174,A 179.99068,B 0.00000,C -180.00000} ; retreat
  ; Step 137, bar 3264
  LIN {X -14736.114,Y -970.921,Z 793.666,A 0.00932,B 0.00000,C 180.00000} ; outside
  LIN {X -14736.114,Y -970.921,Z -168.174,A 0.00932,B 0.00000,C 180.00000} ; preinsert
  LIN {X -14736.114,Y -970.921,Z -418.174,A 0.00932,B 0.00000,C 180.00000} ; insert
  LIN {X -14736.114,Y -970.921,Z -418.174,A 0.00932,B 0.00000,C 180.00000} ; release
  LIN {X -14736.114,Y -970.921,Z -118.174,A 0.00932,B 0.00000,C 180.00000} ; retreat
  ; Step 138, bar 3344
  LIN {X 14736.114,Y -970.921,Z 793.666,A 179.99068,B 0.00000,C 180.00000} ; outside
  LIN {X 14736.114,Y -970.921,Z -168.174,A 179.99068,B 0.00000,C 180.00000} ; preinsert
  LIN {X 14736.114,Y -970.921,Z -418.174,A 179.99068,B 0.00000,C 180.00000} ; insert
  LIN {X 14736.114,Y -970.921,Z -418.174,A 179.99068,B 0.00000,C 180.00000} ; release
  LIN {X 14736.114,Y -970.921,Z -118.174,A 179.99068,B 0.00000,C 180.00000} ; retreat
  ; Step 139, bar 3265
  LIN {X -14736.114,Y -885.921,Z 793.666,A 0.00932,B 0.00000,C 180.00000} ; outside
  LIN {X -14736.114,Y -885.921,Z -168.174,A 0.00932,B 0.00000,C 180.00000} ; preinsert
  LIN {X -14736.114,Y -885.921,Z -418.174,A 0.00932,B 0.00000,C 180.00000} ; insert
  LIN {X -14736.114,Y -885.921,Z -418.174,A 0.00932,B 0.00000,C 180.00000} ; release
  LIN {X -14736.114,Y -885.921,Z -118.174,A 0.00932,B 0.00000,C 180.00000} ; retreat
  ; Step 140, bar 3345
  LIN {X 14736.114,Y -885.921,Z 793.666,A 179.99068,B 0.00000,C 180.00000} ; outside
  LIN {X 14736.114,Y -885.921,Z -168.174,A 179.99068,B 0.00000,C 180.00000} ; preinsert
  LIN {X 14736.114,Y -885.921,Z -418.174,A 179.99068,B 0.00000,C 180.00000} ; insert
  LIN {X 14736.114,Y -885.921,Z -418.174,A 179.99068,B 0.00000,C 180.00000} ; release
  LIN {X 14736.114,Y -885.921,Z -118.174,A 179.99068,B 0.00000,C 180.00000} ; retreat
  ; Step 141, bar 3266
  LIN {X -14736.114,Y -800.921,Z 793.666,A 0.00932,B 0.00000,C 180.00000} ; outside
  LIN {X -14736.114,Y -800.921,Z -168.174,A 0.00932,B 0.00000,C 180.00000} ; preinsert
  LIN {X -14736.114,Y -800.921,Z -418.174,A 0.00932,B 0.00000,C 180.00000} ; insert
  LIN {X -14736.114,Y -800.921,Z -418.174,A 0.00932,B 0.00000,C 180.00000} ; release
  LIN {X -14736.114,Y -800.921,Z -118.174,A 0.00932,B 0.00000,C 180.00000} ; retreat
  ; Step 142, bar 3346
  LIN {X 14736.114,Y -800.921,Z 793.666,A 179.99068,B 0.00000,C 180.00000} ; outside
  LIN {X 14736.114,Y -800.921,Z -168.174,A 179.99068,B 0.00000,C 180.00000} ; preinsert
  LIN {X 14736.114,Y -800.921,Z -418.174,A 179.99068,B 0.00000,C 180.00000} ; insert
  LIN {X 14736.114,Y -800.921,Z -418.174,A 179.99068,B 0.00000,C 180.00000} ; release
  LIN {X 14736.114,Y -800.921,Z -118.174,A 179.99068,B 0.00000,C 180.00000} ; retreat
  ; Step 143, bar 3306
  LIN {X -14736.114,Y 800.921,Z 793.666,A -0.00932,B 0.00000,C 180.00000} ; outside
  LIN {X -14736.114,Y 800.921,Z -168.174,A -0.00932,B 0.00000,C 180.00000} ; preinsert
  LIN {X -14736.114,Y 800.921,Z -418.174,A -0.00932,B 0.00000,C 180.00000} ; insert
  LIN {X -14736.114,Y 800.921,Z -418.174,A -0.00932,B 0.00000,C 180.00000} ; release
  LIN {X -14736.114,Y 800.921,Z -118.174,A -0.00932,B 0.00000,C 180.00000} ; retreat
  ; Step 144, bar 3386
  LIN {X 14736.114,Y 800.921,Z 793.666,A -179.99068,B 0.00000,C -180.00000} ; outside
  LIN {X 14736.114,Y 800.921,Z -168.174,A -179.99068,B 0.00000,C -180.00000} ; preinsert
  LIN {X 14736.114,Y 800.921,Z -418.174,A -179.99068,B 0.00000,C -180.00000} ; insert
  LIN {X 14736.114,Y 800.921,Z -418.174,A -179.99068,B 0.00000,C -180.00000} ; release
  LIN {X 14736.114,Y 800.921,Z -118.174,A -179.99068,B 0.00000,C -180.00000} ; retreat
  ; Step 145, bar 3305
  LIN {X -14736.114,Y 885.921,Z 793.666,A -0.00932,B 0.00000,C 180.00000} ; outside
  LIN {X -14736.114,Y 885.921,Z -168.174,A -0.00932,B 0.00000,C 180.00000} ; preinsert
  LIN {X -14736.114,Y 885.921,Z -418.174,A -0.00932,B 0.00000,C 180.00000} ; insert
  LIN {X -14736.114,Y 885.921,Z -418.174,A -0.00932,B 0.00000,C 180.00000} ; release
  LIN {X -14736.114,Y 885.921,Z -118.174,A -0.00932,B 0.00000,C 180.00000} ; retreat
  ; Step 146, bar 3385
  LIN {X 14736.114,Y 885.921,Z 793.666,A -179.99068,B 0.00000,C -180.00000} ; outside
  LIN {X 14736.114,Y 885.921,Z -168.174,A -179.99068,B 0.00000,C -180.00000} ; preinsert
  LIN {X 14736.114,Y 885.921,Z -418.174,A -179.99068,B 0.00000,C -180.00000} ; insert
  LIN {X 14736.114,Y 885.921,Z -418.174,A -179.99068,B 0.00000,C -180.00000} ; release
  LIN {X 14736.114,Y 885.921,Z -118.174,A -179.99068,B 0.00000,C -180.00000} ; retreat
  ; Step 147, bar 3304
  LIN {X -14736.114,Y 970.921,Z 793.666,A -0.00932,B 0.00000,C 180.00000} ; outside
  LIN {X -14736.114,Y 970.921,Z -168.174,A -0.00932,B 0.00000,C 180.00000} ; preinsert
  LIN {X -14736.114,Y 970.921,Z -418.174,A -0.00932,B 0.00000,C 180.00000} ; insert
  LIN {X -14736.114,Y 970.921,Z -418.174,A -0.00932,B 0.00000,C 180.00000} ; release
  LIN {X -14736.114,Y 970.921,Z -118.174,A -0.00932,B 0.00000,C 180.00000} ; retreat
  ; Step 148, bar 3384
  LIN {X 14736.114,Y 970.921,Z 793.666,A -179.99068,B 0.00000,C -180.00000} ; outside
  LIN {X 14736.114,Y 970.921,Z -168.174,A -179.99068,B 0.00000,C -180.00000} ; preinsert
  LIN {X 14736.114,Y 970.921,Z -418.174,A -179.99068,B 0.00000,C -180.00000} ; insert
  LIN {X 14736.114,Y 970.921,Z -418.174,A -179.99068,B 0.00000,C -180.00000} ; release
  LIN {X 14736.114,Y 970.921,Z -118.174,A -179.99068,B 0.00000,C -180.00000} ; retreat
  ; Step 149, bar 3296
  LIN {X -14736.114,Y 1128.921,Z 793.666,A -0.00932,B 0.00000,C 180.00000} ; outside
  LIN {X -14736.114,Y 1128.921,Z -168.174,A -0.00932,B 0.00000,C 180.00000} ; preinsert
  LIN {X -14736.114,Y 1128.921,Z -418.174,A -0.00932,B 0.00000,C 180.00000} ; insert
  LIN {X -14736.114,Y 1128.921,Z -418.174,A -0.00932,B 0.00000,C 180.00000} ; release
  LIN {X -14736.114,Y 1128.921,Z -118.174,A -0.00932,B 0.00000,C 180.00000} ; retreat
  ; Step 150, bar 3376
  LIN {X 14736.114,Y 1128.921,Z 793.666,A -179.99068,B 0.00000,C -180.00000} ; outside
  LIN {X 14736.114,Y 1128.921,Z -168.174,A -179.99068,B 0.00000,C -180.00000} ; preinsert
  LIN {X 14736.114,Y 1128.921,Z -418.174,A -179.99068,B 0.00000,C -180.00000} ; insert
  LIN {X 14736.114,Y 1128.921,Z -418.174,A -179.99068,B 0.00000,C -180.00000} ; release
  LIN {X 14736.114,Y 1128.921,Z -118.174,A -179.99068,B 0.00000,C -180.00000} ; retreat
  ; Step 151, bar 3307
  LIN {X -14736.114,Y 1213.921,Z 793.666,A -0.00932,B 0.00000,C 180.00000} ; outside
  LIN {X -14736.114,Y 1213.921,Z -168.174,A -0.00932,B 0.00000,C 180.00000} ; preinsert
  LIN {X -14736.114,Y 1213.921,Z -418.174,A -0.00932,B 0.00000,C 180.00000} ; insert
  LIN {X -14736.114,Y 1213.921,Z -418.174,A -0.00932,B 0.00000,C 180.00000} ; release
  LIN {X -14736.114,Y 1213.921,Z -118.174,A -0.00932,B 0.00000,C 180.00000} ; retreat
  ; Step 152, bar 3387
  LIN {X 14736.114,Y 1213.921,Z 793.666,A -179.99068,B 0.00000,C -180.00000} ; outside
  LIN {X 14736.114,Y 1213.921,Z -168.174,A -179.99068,B 0.00000,C -180.00000} ; preinsert
  LIN {X 14736.114,Y 1213.921,Z -418.174,A -179.99068,B 0.00000,C -180.00000} ; insert
  LIN {X 14736.114,Y 1213.921,Z -418.174,A -179.99068,B 0.00000,C -180.00000} ; release
  LIN {X 14736.114,Y 1213.921,Z -118.174,A -179.99068,B 0.00000,C -180.00000} ; retreat
  ; Step 153, bar 3192
  LIN {X -14073.123,Y -2173.194,Z 792.663,A 134.95763,B 0.00000,C 180.00000} ; outside
  LIN {X -14073.123,Y -2173.194,Z -61.962,A 134.95763,B 0.00000,C 180.00000} ; preinsert
  LIN {X -14073.123,Y -2173.194,Z -311.962,A 134.95763,B 0.00000,C 180.00000} ; insert
  LIN {X -14073.123,Y -2173.194,Z -311.962,A 134.95763,B 0.00000,C 180.00000} ; release
  LIN {X -14073.123,Y -2173.194,Z -11.962,A 134.95763,B 0.00000,C 180.00000} ; retreat
  ; Step 154, bar 3194
  LIN {X -13926.877,Y -2173.194,Z 792.663,A 45.04237,B 0.00000,C 180.00000} ; outside
  LIN {X -13926.877,Y -2173.194,Z -61.962,A 45.04237,B 0.00000,C 180.00000} ; preinsert
  LIN {X -13926.877,Y -2173.194,Z -311.962,A 45.04237,B 0.00000,C 180.00000} ; insert
  LIN {X -13926.877,Y -2173.194,Z -311.962,A 45.04237,B 0.00000,C 180.00000} ; release
  LIN {X -13926.877,Y -2173.194,Z -11.962,A 45.04237,B 0.00000,C 180.00000} ; retreat
  ; Step 155, bar 3200
  LIN {X -10073.123,Y -2173.194,Z 792.663,A 134.95763,B 0.00000,C 180.00000} ; outside
  LIN {X -10073.123,Y -2173.194,Z -61.962,A 134.95763,B 0.00000,C 180.00000} ; preinsert
  LIN {X -10073.123,Y -2173.194,Z -311.962,A 134.95763,B 0.00000,C 180.00000} ; insert
  LIN {X -10073.123,Y -2173.194,Z -311.962,A 134.95763,B 0.00000,C 180.00000} ; release
  LIN {X -10073.123,Y -2173.194,Z -11.962,A 134.95763,B 0.00000,C 180.00000} ; retreat
  ; Step 156, bar 3202
  LIN {X -9926.877,Y -2173.194,Z 792.663,A 45.04237,B 0.00000,C 180.00000} ; outside
  LIN {X -9926.877,Y -2173.194,Z -61.962,A 45.04237,B 0.00000,C 180.00000} ; preinsert
  LIN {X -9926.877,Y -2173.194,Z -311.962,A 45.04237,B 0.00000,C 180.00000} ; insert
  LIN {X -9926.877,Y -2173.194,Z -311.962,A 45.04237,B 0.00000,C 180.00000} ; release
  LIN {X -9926.877,Y -2173.194,Z -11.962,A 45.04237,B 0.00000,C 180.00000} ; retreat
  ; Step 157, bar 3208
  LIN {X -6073.123,Y -2173.194,Z 792.663,A 134.95763,B 0.00000,C 180.00000} ; outside
  LIN {X -6073.123,Y -2173.194,Z -61.962,A 134.95763,B 0.00000,C 180.00000} ; preinsert
  LIN {X -6073.123,Y -2173.194,Z -311.962,A 134.95763,B 0.00000,C 180.00000} ; insert
  LIN {X -6073.123,Y -2173.194,Z -311.962,A 134.95763,B 0.00000,C 180.00000} ; release
  LIN {X -6073.123,Y -2173.194,Z -11.962,A 134.95763,B 0.00000,C 180.00000} ; retreat
  ; Step 158, bar 3210
  LIN {X -5926.877,Y -2173.194,Z 792.663,A 45.04237,B 0.00000,C 180.00000} ; outside
  LIN {X -5926.877,Y -2173.194,Z -61.962,A 45.04237,B 0.00000,C 180.00000} ; preinsert
  LIN {X -5926.877,Y -2173.194,Z -311.962,A 45.04237,B 0.00000,C 180.00000} ; insert
  LIN {X -5926.877,Y -2173.194,Z -311.962,A 45.04237,B 0.00000,C 180.00000} ; release
  LIN {X -5926.877,Y -2173.194,Z -11.962,A 45.04237,B 0.00000,C 180.00000} ; retreat
  ; Step 159, bar 3216
  LIN {X -2073.121,Y -2173.194,Z 792.663,A 134.95763,B 0.00000,C -180.00000} ; outside
  LIN {X -2073.121,Y -2173.194,Z -61.962,A 134.95763,B 0.00000,C -180.00000} ; preinsert
  LIN {X -2073.121,Y -2173.194,Z -311.962,A 134.95763,B 0.00000,C -180.00000} ; insert
  LIN {X -2073.121,Y -2173.194,Z -311.962,A 134.95763,B 0.00000,C -180.00000} ; release
  LIN {X -2073.121,Y -2173.194,Z -11.962,A 134.95763,B 0.00000,C -180.00000} ; retreat
  ; Step 160, bar 3218
  LIN {X -1926.875,Y -2173.194,Z 792.663,A 45.04237,B 0.00000,C 180.00000} ; outside
  LIN {X -1926.875,Y -2173.194,Z -61.962,A 45.04237,B 0.00000,C 180.00000} ; preinsert
  LIN {X -1926.875,Y -2173.194,Z -311.962,A 45.04237,B 0.00000,C 180.00000} ; insert
  LIN {X -1926.875,Y -2173.194,Z -311.962,A 45.04237,B 0.00000,C 180.00000} ; release
  LIN {X -1926.875,Y -2173.194,Z -11.962,A 45.04237,B 0.00000,C 180.00000} ; retreat
  ; Step 161, bar 3224
  LIN {X 1926.879,Y -2173.194,Z 792.663,A 134.95763,B 0.00000,C -180.00000} ; outside
  LIN {X 1926.879,Y -2173.194,Z -61.962,A 134.95763,B 0.00000,C -180.00000} ; preinsert
  LIN {X 1926.879,Y -2173.194,Z -311.962,A 134.95763,B 0.00000,C -180.00000} ; insert
  LIN {X 1926.879,Y -2173.194,Z -311.962,A 134.95763,B 0.00000,C -180.00000} ; release
  LIN {X 1926.879,Y -2173.194,Z -11.962,A 134.95763,B 0.00000,C -180.00000} ; retreat
  ; Step 162, bar 3226
  LIN {X 2073.125,Y -2173.194,Z 792.663,A 45.04237,B 0.00000,C 180.00000} ; outside
  LIN {X 2073.125,Y -2173.194,Z -61.962,A 45.04237,B 0.00000,C 180.00000} ; preinsert
  LIN {X 2073.125,Y -2173.194,Z -311.962,A 45.04237,B 0.00000,C 180.00000} ; insert
  LIN {X 2073.125,Y -2173.194,Z -311.962,A 45.04237,B 0.00000,C 180.00000} ; release
  LIN {X 2073.125,Y -2173.194,Z -11.962,A 45.04237,B 0.00000,C 180.00000} ; retreat
  ; Step 163, bar 3232
  LIN {X 5926.879,Y -2173.194,Z 792.663,A 134.95763,B 0.00000,C 180.00000} ; outside
  LIN {X 5926.879,Y -2173.194,Z -61.962,A 134.95763,B 0.00000,C 180.00000} ; preinsert
  LIN {X 5926.879,Y -2173.194,Z -311.962,A 134.95763,B 0.00000,C 180.00000} ; insert
  LIN {X 5926.879,Y -2173.194,Z -311.962,A 134.95763,B 0.00000,C 180.00000} ; release
  LIN {X 5926.879,Y -2173.194,Z -11.962,A 134.95763,B 0.00000,C 180.00000} ; retreat
  ; Step 164, bar 3234
  LIN {X 6073.125,Y -2173.194,Z 792.663,A 45.04237,B 0.00000,C 180.00000} ; outside
  LIN {X 6073.125,Y -2173.194,Z -61.962,A 45.04237,B 0.00000,C 180.00000} ; preinsert
  LIN {X 6073.125,Y -2173.194,Z -311.962,A 45.04237,B 0.00000,C 180.00000} ; insert
  LIN {X 6073.125,Y -2173.194,Z -311.962,A 45.04237,B 0.00000,C 180.00000} ; release
  LIN {X 6073.125,Y -2173.194,Z -11.962,A 45.04237,B 0.00000,C 180.00000} ; retreat
  ; Step 165, bar 3240
  LIN {X 9926.879,Y -2173.194,Z 792.663,A 134.95763,B 0.00000,C 180.00000} ; outside
  LIN {X 9926.879,Y -2173.194,Z -61.962,A 134.95763,B 0.00000,C 180.00000} ; preinsert
  LIN {X 9926.879,Y -2173.194,Z -311.962,A 134.95763,B 0.00000,C 180.00000} ; insert
  LIN {X 9926.879,Y -2173.194,Z -311.962,A 134.95763,B 0.00000,C 180.00000} ; release
  LIN {X 9926.879,Y -2173.194,Z -11.962,A 134.95763,B 0.00000,C 180.00000} ; retreat
  ; Step 166, bar 3242
  LIN {X 10073.125,Y -2173.194,Z 792.663,A 45.04237,B 0.00000,C 180.00000} ; outside
  LIN {X 10073.125,Y -2173.194,Z -61.962,A 45.04237,B 0.00000,C 180.00000} ; preinsert
  LIN {X 10073.125,Y -2173.194,Z -311.962,A 45.04237,B 0.00000,C 180.00000} ; insert
  LIN {X 10073.125,Y -2173.194,Z -311.962,A 45.04237,B 0.00000,C 180.00000} ; release
  LIN {X 10073.125,Y -2173.194,Z -11.962,A 45.04237,B 0.00000,C 180.00000} ; retreat
  ; Step 167, bar 3248
  LIN {X 13926.879,Y -2173.194,Z 792.663,A 134.95763,B 0.00000,C 180.00000} ; outside
  LIN {X 13926.879,Y -2173.194,Z -61.962,A 134.95763,B 0.00000,C 180.00000} ; preinsert
  LIN {X 13926.879,Y -2173.194,Z -311.962,A 134.95763,B 0.00000,C 180.00000} ; insert
  LIN {X 13926.879,Y -2173.194,Z -311.962,A 134.95763,B 0.00000,C 180.00000} ; release
  LIN {X 13926.879,Y -2173.194,Z -11.962,A 134.95763,B 0.00000,C 180.00000} ; retreat
  ; Step 168, bar 3250
  LIN {X 14073.125,Y -2173.194,Z 792.663,A 45.04237,B 0.00000,C 180.00000} ; outside
  LIN {X 14073.125,Y -2173.194,Z -61.962,A 45.04237,B 0.00000,C 180.00000} ; preinsert
  LIN {X 14073.125,Y -2173.194,Z -311.962,A 45.04237,B 0.00000,C 180.00000} ; insert
  LIN {X 14073.125,Y -2173.194,Z -311.962,A 45.04237,B 0.00000,C 180.00000} ; release
  LIN {X 14073.125,Y -2173.194,Z -11.962,A 45.04237,B 0.00000,C 180.00000} ; retreat
  ; Step 169, bar 3193
  LIN {X -14073.194,Y -2026.877,Z 792.663,A 44.95763,B 0.00000,C 180.00000} ; outside
  LIN {X -14073.194,Y -2026.877,Z -61.962,A 44.95763,B 0.00000,C 180.00000} ; preinsert
  LIN {X -14073.194,Y -2026.877,Z -311.962,A 44.95763,B 0.00000,C 180.00000} ; insert
  LIN {X -14073.194,Y -2026.877,Z -311.962,A 44.95763,B 0.00000,C 180.00000} ; release
  LIN {X -14073.194,Y -2026.877,Z -11.962,A 44.95763,B 0.00000,C 180.00000} ; retreat
  ; Step 170, bar 3201
  LIN {X -10073.194,Y -2026.877,Z 792.663,A 44.95763,B 0.00000,C 180.00000} ; outside
  LIN {X -10073.194,Y -2026.877,Z -61.962,A 44.95763,B 0.00000,C 180.00000} ; preinsert
  LIN {X -10073.194,Y -2026.877,Z -311.962,A 44.95763,B 0.00000,C 180.00000} ; insert
  LIN {X -10073.194,Y -2026.877,Z -311.962,A 44.95763,B 0.00000,C 180.00000} ; release
  LIN {X -10073.194,Y -2026.877,Z -11.962,A 44.95763,B 0.00000,C 180.00000} ; retreat
  ; Step 171, bar 3209
  LIN {X -6073.194,Y -2026.877,Z 792.663,A 44.95763,B 0.00000,C 180.00000} ; outside
  LIN {X -6073.194,Y -2026.877,Z -61.962,A 44.95763,B 0.00000,C 180.00000} ; preinsert
  LIN {X -6073.194,Y -2026.877,Z -311.962,A 44.95763,B 0.00000,C 180.00000} ; insert
  LIN {X -6073.194,Y -2026.877,Z -311.962,A 44.95763,B 0.00000,C 180.00000} ; release
  LIN {X -6073.194,Y -2026.877,Z -11.962,A 44.95763,B 0.00000,C 180.00000} ; retreat
  ; Step 172, bar 3217
  LIN {X -2073.193,Y -2026.877,Z 792.663,A 44.95763,B 0.00000,C 180.00000} ; outside
  LIN {X -2073.193,Y -2026.877,Z -61.962,A 44.95763,B 0.00000,C 180.00000} ; preinsert
  LIN {X -2073.193,Y -2026.877,Z -311.962,A 44.95763,B 0.00000,C 180.00000} ; insert
  LIN {X -2073.193,Y -2026.877,Z -311.962,A 44.95763,B 0.00000,C 180.00000} ; release
  LIN {X -2073.193,Y -2026.877,Z -11.962,A 44.95763,B 0.00000,C 180.00000} ; retreat
  ; Step 173, bar 3225
  LIN {X 1926.807,Y -2026.877,Z 792.663,A 44.95763,B 0.00000,C 180.00000} ; outside
  LIN {X 1926.807,Y -2026.877,Z -61.962,A 44.95763,B 0.00000,C 180.00000} ; preinsert
  LIN {X 1926.807,Y -2026.877,Z -311.962,A 44.95763,B 0.00000,C 180.00000} ; insert
  LIN {X 1926.807,Y -2026.877,Z -311.962,A 44.95763,B 0.00000,C 180.00000} ; release
  LIN {X 1926.807,Y -2026.877,Z -11.962,A 44.95763,B 0.00000,C 180.00000} ; retreat
  ; Step 174, bar 3233
  LIN {X 5926.807,Y -2026.877,Z 792.663,A 44.95763,B 0.00000,C 180.00000} ; outside
  LIN {X 5926.807,Y -2026.877,Z -61.962,A 44.95763,B 0.00000,C 180.00000} ; preinsert
  LIN {X 5926.807,Y -2026.877,Z -311.962,A 44.95763,B 0.00000,C 180.00000} ; insert
  LIN {X 5926.807,Y -2026.877,Z -311.962,A 44.95763,B 0.00000,C 180.00000} ; release
  LIN {X 5926.807,Y -2026.877,Z -11.962,A 44.95763,B 0.00000,C 180.00000} ; retreat
  ; Step 175, bar 3241
  LIN {X 9926.807,Y -2026.877,Z 792.663,A 44.95763,B 0.00000,C 180.00000} ; outside
  LIN {X 9926.807,Y -2026.877,Z -61.962,A 44.95763,B 0.00000,C 180.00000} ; preinsert
  LIN {X 9926.807,Y -2026.877,Z -311.962,A 44.95763,B 0.00000,C 180.00000} ; insert
  LIN {X 9926.807,Y -2026.877,Z -311.962,A 44.95763,B 0.00000,C 180.00000} ; release
  LIN {X 9926.807,Y -2026.877,Z -11.962,A 44.95763,B 0.00000,C 180.00000} ; retreat
  ; Step 176, bar 3249
  LIN {X 13926.807,Y -2026.877,Z 792.663,A 44.95763,B 0.00000,C 180.00000} ; outside
  LIN {X 13926.807,Y -2026.877,Z -61.962,A 44.95763,B 0.00000,C 180.00000} ; preinsert
  LIN {X 13926.807,Y -2026.877,Z -311.962,A 44.95763,B 0.00000,C 180.00000} ; insert
  LIN {X 13926.807,Y -2026.877,Z -311.962,A 44.95763,B 0.00000,C 180.00000} ; release
  LIN {X 13926.807,Y -2026.877,Z -11.962,A 44.95763,B 0.00000,C 180.00000} ; retreat
  ; Step 177, bar 3195
  LIN {X -13926.806,Y -2026.877,Z 792.663,A 135.04237,B 0.00000,C 180.00000} ; outside
  LIN {X -13926.806,Y -2026.877,Z -61.962,A 135.04237,B 0.00000,C 180.00000} ; preinsert
  LIN {X -13926.806,Y -2026.877,Z -311.962,A 135.04237,B 0.00000,C 180.00000} ; insert
  LIN {X -13926.806,Y -2026.877,Z -311.962,A 135.04237,B 0.00000,C 180.00000} ; release
  LIN {X -13926.806,Y -2026.877,Z -11.962,A 135.04237,B 0.00000,C 180.00000} ; retreat
  ; Step 178, bar 3203
  LIN {X -9926.806,Y -2026.877,Z 792.663,A 135.04237,B 0.00000,C 180.00000} ; outside
  LIN {X -9926.806,Y -2026.877,Z -61.962,A 135.04237,B 0.00000,C 180.00000} ; preinsert
  LIN {X -9926.806,Y -2026.877,Z -311.962,A 135.04237,B 0.00000,C 180.00000} ; insert
  LIN {X -9926.806,Y -2026.877,Z -311.962,A 135.04237,B 0.00000,C 180.00000} ; release
  LIN {X -9926.806,Y -2026.877,Z -11.962,A 135.04237,B 0.00000,C 180.00000} ; retreat
  ; Step 179, bar 3211
  LIN {X -5926.806,Y -2026.877,Z 792.663,A 135.04237,B 0.00000,C 180.00000} ; outside
  LIN {X -5926.806,Y -2026.877,Z -61.962,A 135.04237,B 0.00000,C 180.00000} ; preinsert
  LIN {X -5926.806,Y -2026.877,Z -311.962,A 135.04237,B 0.00000,C 180.00000} ; insert
  LIN {X -5926.806,Y -2026.877,Z -311.962,A 135.04237,B 0.00000,C 180.00000} ; release
  LIN {X -5926.806,Y -2026.877,Z -11.962,A 135.04237,B 0.00000,C 180.00000} ; retreat
  ; Step 180, bar 3219
  LIN {X -1926.804,Y -2026.877,Z 792.663,A 135.04237,B 0.00000,C 180.00000} ; outside
  LIN {X -1926.804,Y -2026.877,Z -61.962,A 135.04237,B 0.00000,C 180.00000} ; preinsert
  LIN {X -1926.804,Y -2026.877,Z -311.962,A 135.04237,B 0.00000,C 180.00000} ; insert
  LIN {X -1926.804,Y -2026.877,Z -311.962,A 135.04237,B 0.00000,C 180.00000} ; release
  LIN {X -1926.804,Y -2026.877,Z -11.962,A 135.04237,B 0.00000,C 180.00000} ; retreat
  ; Step 181, bar 3227
  LIN {X 2073.196,Y -2026.877,Z 792.663,A 135.04237,B 0.00000,C 180.00000} ; outside
  LIN {X 2073.196,Y -2026.877,Z -61.962,A 135.04237,B 0.00000,C 180.00000} ; preinsert
  LIN {X 2073.196,Y -2026.877,Z -311.962,A 135.04237,B 0.00000,C 180.00000} ; insert
  LIN {X 2073.196,Y -2026.877,Z -311.962,A 135.04237,B 0.00000,C 180.00000} ; release
  LIN {X 2073.196,Y -2026.877,Z -11.962,A 135.04237,B 0.00000,C 180.00000} ; retreat
  ; Step 182, bar 3235
  LIN {X 6073.196,Y -2026.877,Z 792.663,A 135.04237,B 0.00000,C 180.00000} ; outside
  LIN {X 6073.196,Y -2026.877,Z -61.962,A 135.04237,B 0.00000,C 180.00000} ; preinsert
  LIN {X 6073.196,Y -2026.877,Z -311.962,A 135.04237,B 0.00000,C 180.00000} ; insert
  LIN {X 6073.196,Y -2026.877,Z -311.962,A 135.04237,B 0.00000,C 180.00000} ; release
  LIN {X 6073.196,Y -2026.877,Z -11.962,A 135.04237,B 0.00000,C 180.00000} ; retreat
  ; Step 183, bar 3243
  LIN {X 10073.196,Y -2026.877,Z 792.663,A 135.04237,B 0.00000,C 180.00000} ; outside
  LIN {X 10073.196,Y -2026.877,Z -61.962,A 135.04237,B 0.00000,C 180.00000} ; preinsert
  LIN {X 10073.196,Y -2026.877,Z -311.962,A 135.04237,B 0.00000,C 180.00000} ; insert
  LIN {X 10073.196,Y -2026.877,Z -311.962,A 135.04237,B 0.00000,C 180.00000} ; release
  LIN {X 10073.196,Y -2026.877,Z -11.962,A 135.04237,B 0.00000,C 180.00000} ; retreat
  ; Step 184, bar 3251
  LIN {X 14073.196,Y -2026.877,Z 792.663,A 135.04237,B 0.00000,C 180.00000} ; outside
  LIN {X 14073.196,Y -2026.877,Z -61.962,A 135.04237,B 0.00000,C 180.00000} ; preinsert
  LIN {X 14073.196,Y -2026.877,Z -311.962,A 135.04237,B 0.00000,C 180.00000} ; insert
  LIN {X 14073.196,Y -2026.877,Z -311.962,A 135.04237,B 0.00000,C 180.00000} ; release
  LIN {X 14073.196,Y -2026.877,Z -11.962,A 135.04237,B 0.00000,C 180.00000} ; retreat
  ; Step 185, bar 3187
  LIN {X 14073.196,Y 2026.877,Z 792.663,A -135.04237,B 0.00000,C 180.00000} ; outside
  LIN {X 14073.196,Y 2026.877,Z -61.962,A -135.04237,B 0.00000,C 180.00000} ; preinsert
  LIN {X 14073.196,Y 2026.877,Z -311.962,A -135.04237,B 0.00000,C 180.00000} ; insert
  LIN {X 14073.196,Y 2026.877,Z -311.962,A -135.04237,B 0.00000,C 180.00000} ; release
  LIN {X 14073.196,Y 2026.877,Z -11.962,A -135.04237,B 0.00000,C 180.00000} ; retreat
  ; Step 186, bar 3179
  LIN {X 10073.196,Y 2026.877,Z 792.663,A -135.04237,B 0.00000,C 180.00000} ; outside
  LIN {X 10073.196,Y 2026.877,Z -61.962,A -135.04237,B 0.00000,C 180.00000} ; preinsert
  LIN {X 10073.196,Y 2026.877,Z -311.962,A -135.04237,B 0.00000,C 180.00000} ; insert
  LIN {X 10073.196,Y 2026.877,Z -311.962,A -135.04237,B 0.00000,C 180.00000} ; release
  LIN {X 10073.196,Y 2026.877,Z -11.962,A -135.04237,B 0.00000,C 180.00000} ; retreat
  ; Step 187, bar 3171
  LIN {X 6073.196,Y 2026.877,Z 792.663,A -135.04237,B 0.00000,C -180.00000} ; outside
  LIN {X 6073.196,Y 2026.877,Z -61.962,A -135.04237,B 0.00000,C -180.00000} ; preinsert
  LIN {X 6073.196,Y 2026.877,Z -311.962,A -135.04237,B 0.00000,C -180.00000} ; insert
  LIN {X 6073.196,Y 2026.877,Z -311.962,A -135.04237,B 0.00000,C -180.00000} ; release
  LIN {X 6073.196,Y 2026.877,Z -11.962,A -135.04237,B 0.00000,C -180.00000} ; retreat
  ; Step 188, bar 3163
  LIN {X 2073.196,Y 2026.877,Z 792.663,A -135.04237,B 0.00000,C -180.00000} ; outside
  LIN {X 2073.196,Y 2026.877,Z -61.962,A -135.04237,B 0.00000,C -180.00000} ; preinsert
  LIN {X 2073.196,Y 2026.877,Z -311.962,A -135.04237,B 0.00000,C -180.00000} ; insert
  LIN {X 2073.196,Y 2026.877,Z -311.962,A -135.04237,B 0.00000,C -180.00000} ; release
  LIN {X 2073.196,Y 2026.877,Z -11.962,A -135.04237,B 0.00000,C -180.00000} ; retreat
  ; Step 189, bar 3155
  LIN {X -1926.804,Y 2026.877,Z 792.663,A -135.04237,B 0.00000,C -180.00000} ; outside
  LIN {X -1926.804,Y 2026.877,Z -61.962,A -135.04237,B 0.00000,C -180.00000} ; preinsert
  LIN {X -1926.804,Y 2026.877,Z -311.962,A -135.04237,B 0.00000,C -180.00000} ; insert
  LIN {X -1926.804,Y 2026.877,Z -311.962,A -135.04237,B 0.00000,C -180.00000} ; release
  LIN {X -1926.804,Y 2026.877,Z -11.962,A -135.04237,B 0.00000,C -180.00000} ; retreat
  ; Step 190, bar 3147
  LIN {X -5926.806,Y 2026.877,Z 792.663,A -135.04237,B 0.00000,C -180.00000} ; outside
  LIN {X -5926.806,Y 2026.877,Z -61.962,A -135.04237,B 0.00000,C -180.00000} ; preinsert
  LIN {X -5926.806,Y 2026.877,Z -311.962,A -135.04237,B 0.00000,C -180.00000} ; insert
  LIN {X -5926.806,Y 2026.877,Z -311.962,A -135.04237,B 0.00000,C -180.00000} ; release
  LIN {X -5926.806,Y 2026.877,Z -11.962,A -135.04237,B 0.00000,C -180.00000} ; retreat
  ; Step 191, bar 3139
  LIN {X -9926.806,Y 2026.877,Z 792.663,A -135.04237,B 0.00000,C -180.00000} ; outside
  LIN {X -9926.806,Y 2026.877,Z -61.962,A -135.04237,B 0.00000,C -180.00000} ; preinsert
  LIN {X -9926.806,Y 2026.877,Z -311.962,A -135.04237,B 0.00000,C -180.00000} ; insert
  LIN {X -9926.806,Y 2026.877,Z -311.962,A -135.04237,B 0.00000,C -180.00000} ; release
  LIN {X -9926.806,Y 2026.877,Z -11.962,A -135.04237,B 0.00000,C -180.00000} ; retreat
  ; Step 192, bar 3131
  LIN {X -13926.806,Y 2026.877,Z 792.663,A -135.04237,B 0.00000,C 180.00000} ; outside
  LIN {X -13926.806,Y 2026.877,Z -61.962,A -135.04237,B 0.00000,C 180.00000} ; preinsert
  LIN {X -13926.806,Y 2026.877,Z -311.962,A -135.04237,B 0.00000,C 180.00000} ; insert
  LIN {X -13926.806,Y 2026.877,Z -311.962,A -135.04237,B 0.00000,C 180.00000} ; release
  LIN {X -13926.806,Y 2026.877,Z -11.962,A -135.04237,B 0.00000,C 180.00000} ; retreat
  ; Step 193, bar 3185
  LIN {X 13926.808,Y 2026.877,Z 792.663,A -44.95763,B 0.00000,C 180.00000} ; outside
  LIN {X 13926.808,Y 2026.877,Z -61.962,A -44.95763,B 0.00000,C 180.00000} ; preinsert
  LIN {X 13926.808,Y 2026.877,Z -311.962,A -44.95763,B 0.00000,C 180.00000} ; insert
  LIN {X 13926.808,Y 2026.877,Z -311.962,A -44.95763,B 0.00000,C 180.00000} ; release
  LIN {X 13926.808,Y 2026.877,Z -11.962,A -44.95763,B 0.00000,C 180.00000} ; retreat
  ; Step 194, bar 3177
  LIN {X 9926.808,Y 2026.877,Z 792.663,A -44.95763,B 0.00000,C 180.00000} ; outside
  LIN {X 9926.808,Y 2026.877,Z -61.962,A -44.95763,B 0.00000,C 180.00000} ; preinsert
  LIN {X 9926.808,Y 2026.877,Z -311.962,A -44.95763,B 0.00000,C 180.00000} ; insert
  LIN {X 9926.808,Y 2026.877,Z -311.962,A -44.95763,B 0.00000,C 180.00000} ; release
  LIN {X 9926.808,Y 2026.877,Z -11.962,A -44.95763,B 0.00000,C 180.00000} ; retreat
  ; Step 195, bar 3169
  LIN {X 5926.808,Y 2026.877,Z 792.663,A -44.95763,B 0.00000,C 180.00000} ; outside
  LIN {X 5926.808,Y 2026.877,Z -61.962,A -44.95763,B 0.00000,C 180.00000} ; preinsert
  LIN {X 5926.808,Y 2026.877,Z -311.962,A -44.95763,B 0.00000,C 180.00000} ; insert
  LIN {X 5926.808,Y 2026.877,Z -311.962,A -44.95763,B 0.00000,C 180.00000} ; release
  LIN {X 5926.808,Y 2026.877,Z -11.962,A -44.95763,B 0.00000,C 180.00000} ; retreat
  ; Step 196, bar 3161
  LIN {X 1926.808,Y 2026.877,Z 792.663,A -44.95763,B 0.00000,C 180.00000} ; outside
  LIN {X 1926.808,Y 2026.877,Z -61.962,A -44.95763,B 0.00000,C 180.00000} ; preinsert
  LIN {X 1926.808,Y 2026.877,Z -311.962,A -44.95763,B 0.00000,C 180.00000} ; insert
  LIN {X 1926.808,Y 2026.877,Z -311.962,A -44.95763,B 0.00000,C 180.00000} ; release
  LIN {X 1926.808,Y 2026.877,Z -11.962,A -44.95763,B 0.00000,C 180.00000} ; retreat
  ; Step 197, bar 3153
  LIN {X -2073.192,Y 2026.877,Z 792.663,A -44.95763,B 0.00000,C 180.00000} ; outside
  LIN {X -2073.192,Y 2026.877,Z -61.962,A -44.95763,B 0.00000,C 180.00000} ; preinsert
  LIN {X -2073.192,Y 2026.877,Z -311.962,A -44.95763,B 0.00000,C 180.00000} ; insert
  LIN {X -2073.192,Y 2026.877,Z -311.962,A -44.95763,B 0.00000,C 180.00000} ; release
  LIN {X -2073.192,Y 2026.877,Z -11.962,A -44.95763,B 0.00000,C 180.00000} ; retreat
  ; Step 198, bar 3145
  LIN {X -6073.194,Y 2026.877,Z 792.663,A -44.95763,B 0.00000,C 180.00000} ; outside
  LIN {X -6073.194,Y 2026.877,Z -61.962,A -44.95763,B 0.00000,C 180.00000} ; preinsert
  LIN {X -6073.194,Y 2026.877,Z -311.962,A -44.95763,B 0.00000,C 180.00000} ; insert
  LIN {X -6073.194,Y 2026.877,Z -311.962,A -44.95763,B 0.00000,C 180.00000} ; release
  LIN {X -6073.194,Y 2026.877,Z -11.962,A -44.95763,B 0.00000,C 180.00000} ; retreat
  ; Step 199, bar 3137
  LIN {X -10073.194,Y 2026.877,Z 792.663,A -44.95763,B 0.00000,C 180.00000} ; outside
  LIN {X -10073.194,Y 2026.877,Z -61.962,A -44.95763,B 0.00000,C 180.00000} ; preinsert
  LIN {X -10073.194,Y 2026.877,Z -311.962,A -44.95763,B 0.00000,C 180.00000} ; insert
  LIN {X -10073.194,Y 2026.877,Z -311.962,A -44.95763,B 0.00000,C 180.00000} ; release
  LIN {X -10073.194,Y 2026.877,Z -11.962,A -44.95763,B 0.00000,C 180.00000} ; retreat
  ; Step 200, bar 3129
  LIN {X -14073.194,Y 2026.877,Z 792.663,A -44.95763,B 0.00000,C 180.00000} ; outside
  LIN {X -14073.194,Y 2026.877,Z -61.962,A -44.95763,B 0.00000,C 180.00000} ; preinsert
  LIN {X -14073.194,Y 2026.877,Z -311.962,A -44.95763,B 0.00000,C 180.00000} ; insert
  LIN {X -14073.194,Y 2026.877,Z -311.962,A -44.95763,B 0.00000,C 180.00000} ; release
  LIN {X -14073.194,Y 2026.877,Z -11.962,A -44.95763,B 0.00000,C 180.00000} ; retreat
  ; Step 201, bar 3186
  LIN {X 14073.125,Y 2173.194,Z 792.663,A -45.04237,B 0.00000,C 180.00000} ; outside
  LIN {X 14073.125,Y 2173.194,Z -61.962,A -45.04237,B 0.00000,C 180.00000} ; preinsert
  LIN {X 14073.125,Y 2173.194,Z -311.962,A -45.04237,B 0.00000,C 180.00000} ; insert
  LIN {X 14073.125,Y 2173.194,Z -311.962,A -45.04237,B 0.00000,C 180.00000} ; release
  LIN {X 14073.125,Y 2173.194,Z -11.962,A -45.04237,B 0.00000,C 180.00000} ; retreat
  ; Step 202, bar 3184
  LIN {X 13926.879,Y 2173.194,Z 792.663,A -134.95763,B 0.00000,C -180.00000} ; outside
  LIN {X 13926.879,Y 2173.194,Z -61.962,A -134.95763,B 0.00000,C -180.00000} ; preinsert
  LIN {X 13926.879,Y 2173.194,Z -311.962,A -134.95763,B 0.00000,C -180.00000} ; insert
  LIN {X 13926.879,Y 2173.194,Z -311.962,A -134.95763,B 0.00000,C -180.00000} ; release
  LIN {X 13926.879,Y 2173.194,Z -11.962,A -134.95763,B 0.00000,C -180.00000} ; retreat
  ; Step 203, bar 3178
  LIN {X 10073.125,Y 2173.194,Z 792.663,A -45.04237,B 0.00000,C 180.00000} ; outside
  LIN {X 10073.125,Y 2173.194,Z -61.962,A -45.04237,B 0.00000,C 180.00000} ; preinsert
  LIN {X 10073.125,Y 2173.194,Z -311.962,A -45.04237,B 0.00000,C 180.00000} ; insert
  LIN {X 10073.125,Y 2173.194,Z -311.962,A -45.04237,B 0.00000,C 180.00000} ; release
  LIN {X 10073.125,Y 2173.194,Z -11.962,A -45.04237,B 0.00000,C 180.00000} ; retreat
  ; Step 204, bar 3176
  LIN {X 9926.879,Y 2173.194,Z 792.663,A -134.95763,B 0.00000,C -180.00000} ; outside
  LIN {X 9926.879,Y 2173.194,Z -61.962,A -134.95763,B 0.00000,C -180.00000} ; preinsert
  LIN {X 9926.879,Y 2173.194,Z -311.962,A -134.95763,B 0.00000,C -180.00000} ; insert
  LIN {X 9926.879,Y 2173.194,Z -311.962,A -134.95763,B 0.00000,C -180.00000} ; release
  LIN {X 9926.879,Y 2173.194,Z -11.962,A -134.95763,B 0.00000,C -180.00000} ; retreat
  ; Step 205, bar 3170
  LIN {X 6073.125,Y 2173.194,Z 792.663,A -45.04237,B 0.00000,C 180.00000} ; outside
  LIN {X 6073.125,Y 2173.194,Z -61.962,A -45.04237,B 0.00000,C 180.00000} ; preinsert
  LIN {X 6073.125,Y 2173.194,Z -311.962,A -45.04237,B 0.00000,C 180.00000} ; insert
  LIN {X 6073.125,Y 2173.194,Z -311.962,A -45.04237,B 0.00000,C 180.00000} ; release
  LIN {X 6073.125,Y 2173.194,Z -11.962,A -45.04237,B 0.00000,C 180.00000} ; retreat
  ; Step 206, bar 3168
  LIN {X 5926.879,Y 2173.194,Z 792.663,A -134.95763,B 0.00000,C -180.00000} ; outside
  LIN {X 5926.879,Y 2173.194,Z -61.962,A -134.95763,B 0.00000,C -180.00000} ; preinsert
  LIN {X 5926.879,Y 2173.194,Z -311.962,A -134.95763,B 0.00000,C -180.00000} ; insert
  LIN {X 5926.879,Y 2173.194,Z -311.962,A -134.95763,B 0.00000,C -180.00000} ; release
  LIN {X 5926.879,Y 2173.194,Z -11.962,A -134.95763,B 0.00000,C -180.00000} ; retreat
  ; Step 207, bar 3162
  LIN {X 2073.125,Y 2173.194,Z 792.663,A -45.04237,B 0.00000,C 180.00000} ; outside
  LIN {X 2073.125,Y 2173.194,Z -61.962,A -45.04237,B 0.00000,C 180.00000} ; preinsert
  LIN {X 2073.125,Y 2173.194,Z -311.962,A -45.04237,B 0.00000,C 180.00000} ; insert
  LIN {X 2073.125,Y 2173.194,Z -311.962,A -45.04237,B 0.00000,C 180.00000} ; release
  LIN {X 2073.125,Y 2173.194,Z -11.962,A -45.04237,B 0.00000,C 180.00000} ; retreat
  ; Step 208, bar 3160
  LIN {X 1926.879,Y 2173.194,Z 792.663,A -134.95763,B 0.00000,C -180.00000} ; outside
  LIN {X 1926.879,Y 2173.194,Z -61.962,A -134.95763,B 0.00000,C -180.00000} ; preinsert
  LIN {X 1926.879,Y 2173.194,Z -311.962,A -134.95763,B 0.00000,C -180.00000} ; insert
  LIN {X 1926.879,Y 2173.194,Z -311.962,A -134.95763,B 0.00000,C -180.00000} ; release
  LIN {X 1926.879,Y 2173.194,Z -11.962,A -134.95763,B 0.00000,C -180.00000} ; retreat
  ; Step 209, bar 3154
  LIN {X -1926.875,Y 2173.194,Z 792.663,A -45.04237,B 0.00000,C 180.00000} ; outside
  LIN {X -1926.875,Y 2173.194,Z -61.962,A -45.04237,B 0.00000,C 180.00000} ; preinsert
  LIN {X -1926.875,Y 2173.194,Z -311.962,A -45.04237,B 0.00000,C 180.00000} ; insert
  LIN {X -1926.875,Y 2173.194,Z -311.962,A -45.04237,B 0.00000,C 180.00000} ; release
  LIN {X -1926.875,Y 2173.194,Z -11.962,A -45.04237,B 0.00000,C 180.00000} ; retreat
  ; Step 210, bar 3152
  LIN {X -2073.121,Y 2173.194,Z 792.663,A -134.95763,B 0.00000,C -180.00000} ; outside
  LIN {X -2073.121,Y 2173.194,Z -61.962,A -134.95763,B 0.00000,C -180.00000} ; preinsert
  LIN {X -2073.121,Y 2173.194,Z -311.962,A -134.95763,B 0.00000,C -180.00000} ; insert
  LIN {X -2073.121,Y 2173.194,Z -311.962,A -134.95763,B 0.00000,C -180.00000} ; release
  LIN {X -2073.121,Y 2173.194,Z -11.962,A -134.95763,B 0.00000,C -180.00000} ; retreat
  ; Step 211, bar 3146
  LIN {X -5926.877,Y 2173.194,Z 792.663,A -45.04237,B 0.00000,C 180.00000} ; outside
  LIN {X -5926.877,Y 2173.194,Z -61.962,A -45.04237,B 0.00000,C 180.00000} ; preinsert
  LIN {X -5926.877,Y 2173.194,Z -311.962,A -45.04237,B 0.00000,C 180.00000} ; insert
  LIN {X -5926.877,Y 2173.194,Z -311.962,A -45.04237,B 0.00000,C 180.00000} ; release
  LIN {X -5926.877,Y 2173.194,Z -11.962,A -45.04237,B 0.00000,C 180.00000} ; retreat
  ; Step 212, bar 3144
  LIN {X -6073.123,Y 2173.194,Z 792.663,A -134.95763,B 0.00000,C -180.00000} ; outside
  LIN {X -6073.123,Y 2173.194,Z -61.962,A -134.95763,B 0.00000,C -180.00000} ; preinsert
  LIN {X -6073.123,Y 2173.194,Z -311.962,A -134.95763,B 0.00000,C -180.00000} ; insert
  LIN {X -6073.123,Y 2173.194,Z -311.962,A -134.95763,B 0.00000,C -180.00000} ; release
  LIN {X -6073.123,Y 2173.194,Z -11.962,A -134.95763,B 0.00000,C -180.00000} ; retreat
  ; Step 213, bar 3138
  LIN {X -9926.877,Y 2173.194,Z 792.663,A -45.04237,B 0.00000,C 180.00000} ; outside
  LIN {X -9926.877,Y 2173.194,Z -61.962,A -45.04237,B 0.00000,C 180.00000} ; preinsert
  LIN {X -9926.877,Y 2173.194,Z -311.962,A -45.04237,B 0.00000,C 180.00000} ; insert
  LIN {X -9926.877,Y 2173.194,Z -311.962,A -45.04237,B 0.00000,C 180.00000} ; release
  LIN {X -9926.877,Y 2173.194,Z -11.962,A -45.04237,B 0.00000,C 180.00000} ; retreat
  ; Step 214, bar 3136
  LIN {X -10073.123,Y 2173.194,Z 792.663,A -134.95763,B 0.00000,C -180.00000} ; outside
  LIN {X -10073.123,Y 2173.194,Z -61.962,A -134.95763,B 0.00000,C -180.00000} ; preinsert
  LIN {X -10073.123,Y 2173.194,Z -311.962,A -134.95763,B 0.00000,C -180.00000} ; insert
  LIN {X -10073.123,Y 2173.194,Z -311.962,A -134.95763,B 0.00000,C -180.00000} ; release
  LIN {X -10073.123,Y 2173.194,Z -11.962,A -134.95763,B 0.00000,C -180.00000} ; retreat
  ; Step 215, bar 3130
  LIN {X -13926.877,Y 2173.194,Z 792.663,A -45.04237,B 0.00000,C 180.00000} ; outside
  LIN {X -13926.877,Y 2173.194,Z -61.962,A -45.04237,B 0.00000,C 180.00000} ; preinsert
  LIN {X -13926.877,Y 2173.194,Z -311.962,A -45.04237,B 0.00000,C 180.00000} ; insert
  LIN {X -13926.877,Y 2173.194,Z -311.962,A -45.04237,B 0.00000,C 180.00000} ; release
  LIN {X -13926.877,Y 2173.194,Z -11.962,A -45.04237,B 0.00000,C 180.00000} ; retreat
  ; Step 216, bar 3128
  LIN {X -14073.123,Y 2173.194,Z 792.663,A -134.95763,B 0.00000,C -180.00000} ; outside
  LIN {X -14073.123,Y 2173.194,Z -61.962,A -134.95763,B 0.00000,C -180.00000} ; preinsert
  LIN {X -14073.123,Y 2173.194,Z -311.962,A -134.95763,B 0.00000,C -180.00000} ; insert
  LIN {X -14073.123,Y 2173.194,Z -311.962,A -134.95763,B 0.00000,C -180.00000} ; release
  LIN {X -14073.123,Y 2173.194,Z -11.962,A -134.95763,B 0.00000,C -180.00000} ; retreat
  ; Step 217, bar 1864
  LIN {X 0.000,Y -2589.855,Z 792.630,A 0.00000,B 0.00000,C 180.00000} ; outside
  LIN {X 0.000,Y -2589.855,Z -54.271,A 0.00000,B 0.00000,C 180.00000} ; preinsert
  LIN {X 0.000,Y -2589.855,Z -304.271,A 0.00000,B 0.00000,C 180.00000} ; insert
  LIN {X 0.000,Y -2589.855,Z -304.271,A 0.00000,B 0.00000,C 180.00000} ; release
  LIN {X 0.000,Y -2589.855,Z -4.271,A 0.00000,B 0.00000,C 180.00000} ; retreat
  ; Step 218, bar 1877
  LIN {X 0.000,Y 2589.855,Z 792.630,A 0.00000,B 0.00000,C 180.00000} ; outside
  LIN {X 0.000,Y 2589.855,Z -54.271,A 0.00000,B 0.00000,C 180.00000} ; preinsert
  LIN {X 0.000,Y 2589.855,Z -304.271,A 0.00000,B 0.00000,C 180.00000} ; insert
  LIN {X 0.000,Y 2589.855,Z -304.271,A 0.00000,B 0.00000,C 180.00000} ; release
  LIN {X 0.000,Y 2589.855,Z -4.271,A 0.00000,B 0.00000,C 180.00000} ; retreat
  ; Step 219, bar 1951
  LIN {X 0.000,Y -1200.000,Z 792.630,A 0.00000,B 0.00000,C 180.00000} ; outside
  LIN {X 0.000,Y -1200.000,Z -50.063,A 0.00000,B 0.00000,C 180.00000} ; preinsert
  LIN {X 0.000,Y -1200.000,Z -300.063,A 0.00000,B 0.00000,C 180.00000} ; insert
  LIN {X 0.000,Y -1200.000,Z -300.063,A 0.00000,B 0.00000,C 180.00000} ; release
  LIN {X 0.000,Y -1200.000,Z -0.063,A 0.00000,B 0.00000,C 180.00000} ; retreat
  ; Step 220, bar 1946
  LIN {X 0.000,Y 1200.000,Z 792.630,A 0.00000,B 0.00000,C 180.00000} ; outside
  LIN {X 0.000,Y 1200.000,Z -50.063,A 0.00000,B 0.00000,C 180.00000} ; preinsert
  LIN {X 0.000,Y 1200.000,Z -300.063,A 0.00000,B 0.00000,C 180.00000} ; insert
  LIN {X 0.000,Y 1200.000,Z -300.063,A 0.00000,B 0.00000,C 180.00000} ; release
  LIN {X 0.000,Y 1200.000,Z -0.063,A 0.00000,B 0.00000,C 180.00000} ; retreat
  ; Step 221, bar 3423
  LIN {X -16169.500,Y -1557.401,Z 792.630,A 90.00000,B 0.00000,C 180.00000} ; outside
  LIN {X -16169.500,Y -1557.401,Z -42.000,A 90.00000,B 0.00000,C 180.00000} ; preinsert
  LIN {X -16169.500,Y -1557.401,Z -292.000,A 90.00000,B 0.00000,C 180.00000} ; insert
  LIN {X -16169.500,Y -1557.401,Z -292.000,A 90.00000,B 0.00000,C 180.00000} ; release
